TYPE "UDT_UPSMACHSTAT"
TITLE = UDT_MACHSTAT
VERSION : 0.1
//User-defined structure of UPS machine statuses.
   STRUCT
      OpsNormal : Struct   // Ops/Normal
         StopMCP : Bool;   // Byte 1, Bit 0 - Operator Stop MCP Panel
         StopRemoteCon1 : Bool;   // Byte 1, Bit 1 - Operator Stop Remote Console 1
         StopRemoteCon2 : Bool;   // Byte 1, Bit 2 - Operator Stop Remote Console 2
         BuildingStop : Bool;   // Byte 1, Bit 3 - Building Stop via HMI
         BuildingBreak : Bool;   // Byte 1, Bit 4 - Building Break Time via HMI
         PowerSaveShutdown : Bool;   // Byte 1, Bit 5 - Power Save Shutdown
         SorterNotAtSpeed : Bool;   // Byte 1, Bit 6 - Sorter Not at speed
         MaintenanceSysMode : Bool;   // Byte 1, Bit 7 - System in Maintenance Mode
         Spare_8 : Bool;   // Byte 2, Bit 8 - Future / or Machine Specific (To be identyfied)
         Spare_9 : Bool;   // Byte 2, Bit 9 - Future / or Machine Specific (To be identyfied)
         Spare_10 : Bool;   // Byte 2, Bit 10 - Future / or Machine Specific (To be identyfied)
         Spare_11 : Bool;   // Byte 2, Bit 11 - Future / or Machine Specific (To be identyfied)
         Spare_12 : Bool;   // Byte 2, Bit 12 - Future / or Machine Specific (To be identyfied)
         Spare_13 : Bool;   // Byte 2, Bit 13 - Future / or Machine Specific (To be identyfied)
         Spare_14 : Bool;   // Byte 2, Bit 14 - Future / or Machine Specific (To be identyfied)
         Spare_15 : Bool;   // Byte 2, Bit 15 - Future / or Machine Specific (To be identyfied)
         Spare_16 : Bool;   // Byte 3, Bit 16 - Future / or Machine Specific (To be identyfied)
         Spare_17 : Bool;   // Byte 3, Bit 17 - Future / or Machine Specific (To be identyfied)
         Spare_18 : Bool;   // Byte 3, Bit 18 - Future / or Machine Specific (To be identyfied)
         Spare_19 : Bool;   // Byte 3, Bit 19 - Future / or Machine Specific (To be identyfied)
         Spare_20 : Bool;   // Byte 3, Bit 20 - Future / or Machine Specific (To be identyfied)
         Spare_21 : Bool;   // Byte 3, Bit 21 - Future / or Machine Specific (To be identyfied)
         Spare_22 : Bool;   // Byte 3, Bit 22 - Future / or Machine Specific (To be identyfied)
         Spare_23 : Bool;   // Byte 3, Bit 23 - Future / or Machine Specific (To be identyfied)
         Spare_24 : Bool;   // Byte 4, Bit 24 - Future / or Machine Specific (To be identyfied)
         Spare_25 : Bool;   // Byte 4, Bit 25 - Future / or Machine Specific (To be identyfied)
         Spare_26 : Bool;   // Byte 4, Bit 26 - Future / or Machine Specific (To be identyfied)
         Spare_27 : Bool;   // Byte 4, Bit 27 - Future / or Machine Specific (To be identyfied)
         Spare_28 : Bool;   // Byte 4, Bit 28 - Future / or Machine Specific (To be identyfied)
         Spare_29 : Bool;   // Byte 4, Bit 29 - Future / or Machine Specific (To be identyfied)
         Spare_30 : Bool;   // Byte 4, Bit 30 - Future / or Machine Specific (To be identyfied)
         Spare_31 : Bool;   // Byte 4, Bit 31 - Future / or Machine Specific (To be identyfied)
      END_STRUCT;
      SafetyFaults : Struct   // Safety faults
         BuildingEStop : Bool;   // Byte 5, Bit 0 - Building Emergency Stop
         SystemEStop : Bool;   // Byte 5, Bit 1 - System Emergency Stop
         EmerPullCord : Bool;   // Byte 5, Bit 2 - Emergency Pull Cord
         PhotoEyeBlock1 : Bool;   // Byte 5, Bit 3 - Safety Photo Eye Blocked (Long Range Photo Eye) 1
         PlatformLockout1 : Bool;   // Byte 5, Bit 4 - Platform Lockout 1
         PlatformLockout2 : Bool;   // Byte 5, Bit 5 - Platform Lockout 2
         PhotoEyeBlock2 : Bool;   // Byte 5, Bit 6 - Safety Photo Eye Blocked (Long Range Photo Eye) 2
         PhotoEyeBlock3 : Bool;   // Byte 5, Bit 7 - Safety Photo Eye Blocked (Long Range Photo Eye) 3
         Spare_8 : Bool;   // Byte 6, Bit 8 - Future / or Machine Specific (To be identyfied)
         Spare_9 : Bool;   // Byte 6, Bit 9 - Future / or Machine Specific (To be identyfied)
         Spare_10 : Bool;   // Byte 6, Bit 10 - Future / or Machine Specific (To be identyfied)
         Spare_11 : Bool;   // Byte 6, Bit 11 - Future / or Machine Specific (To be identyfied)
         Spare_12 : Bool;   // Byte 6, Bit 12 - Future / or Machine Specific (To be identyfied)
         Spare_13 : Bool;   // Byte 6, Bit 13 - Future / or Machine Specific (To be identyfied)
         Spare_14 : Bool;   // Byte 6, Bit 14 - Future / or Machine Specific (To be identyfied)
         Spare_15 : Bool;   // Byte 6, Bit 15 - Future / or Machine Specific (To be identyfied)
         Spare_16 : Bool;   // Byte 7, Bit 16 - Future / or Machine Specific (To be identyfied)
         Spare_17 : Bool;   // Byte 7, Bit 17 - Future / or Machine Specific (To be identyfied)
         Spare_18 : Bool;   // Byte 7, Bit 18 - Future / or Machine Specific (To be identyfied)
         Spare_19 : Bool;   // Byte 7, Bit 19 - Future / or Machine Specific (To be identyfied)
         Spare_20 : Bool;   // Byte 7, Bit 20 - Future / or Machine Specific (To be identyfied)
         Spare_21 : Bool;   // Byte 7, Bit 21 - Future / or Machine Specific (To be identyfied)
         Spare_22 : Bool;   // Byte 7, Bit 22 - Future / or Machine Specific (To be identyfied)
         Spare_23 : Bool;   // Byte 7, Bit 23 - Future / or Machine Specific (To be identyfied)
         Spare_24 : Bool;   // Byte 8, Bit 24 - Future / or Machine Specific (To be identyfied)
         Spare_25 : Bool;   // Byte 8, Bit 25 - Future / or Machine Specific (To be identyfied)
         Spare_26 : Bool;   // Byte 8, Bit 26 - Future / or Machine Specific (To be identyfied)
         Spare_27 : Bool;   // Byte 8, Bit 27 - Future / or Machine Specific (To be identyfied)
         Spare_28 : Bool;   // Byte 8, Bit 28 - Future / or Machine Specific (To be identyfied)
         Spare_29 : Bool;   // Byte 8, Bit 29 - Future / or Machine Specific (To be identyfied)
         Spare_30 : Bool;   // Byte 8, Bit 30 - Future / or Machine Specific (To be identyfied)
         Spare_31 : Bool;   // Byte 8, Bit 31 - Future / or Machine Specific (To be identyfied)
      END_STRUCT;
      SystemFaults : Struct   // System faults
         PLCRackFault : Bool;   // Byte 9, Bit 0 - PLC Rack Fault
         EncoderFault : Bool;   // Byte 9, Bit 1 - Encoder Fault
         TipperOrDiverterFault : Bool;   // Byte 9, Bit 2 - Tipper / Diverter Fault
         TCPConFail : Bool;   // Byte 9, Bit 3 - TCP Connection Failure
         SensorJam : Bool;   // Byte 9, Bit 4 - Package Detect Sensor Jam
         CamOrScanFail : Bool;   // Byte 9, Bit 5 - Camera / Scanner Failure
         InductPEJam : Bool;   // Byte 9, Bit 6 - Induct Photo Eye Jam
         SortVerificationPEJam : Bool;   // Byte 9, Bit 7 - Sort Verification Photo Eye Jam
         TakeAwayConvPEJam : Bool;   // Byte 10, Bit 8 - Take Away Conveyor Photo Eye Jam
         SorterMechFault : Bool;   // Byte 10, Bit 9 - Sorter Mechanical Fault
         Spare_10 : Bool;   // Byte 10, Bit 10 - Future / or Machine Specific (To be identyfied)
         SorterJam : Bool;   // Byte 10, Bit 11 - Sorter Jam (Logical Failure)
         InductPCAlignmentError : Bool;   // Byte 10, Bit 12 - Induct Photo Cell Alignment Error
         MotorFault : Bool;   // Byte 10, Bit 13 - Motor Fault
         PowerFault : Bool;   // Byte 10, Bit 14 - Power Fault
         Spare_15 : Bool;   // Byte 10, Bit 15 - Future / or Machine Specific (To be identyfied)
         IOComError : Bool;   // Byte 11, Bit 16 - I/O Communications Error
         RemoteIOComError : Bool;   // Byte 11, Bit 17 - Remote I/O Communications Error
         XLeChatComError : Bool;   // Byte 11, Bit 18 - XLe chat Communications Error
         SerialComError : Bool;   // Byte 11, Bit 19 - Serial Communications Error
         SubsystemError : Bool;   // Byte 11, Bit 20 - Subsytem Error (Scale, Camera, etc...)
         VDFFault : Bool;   // Byte 11, Bit 21 - VDF Fault
         SystemResetInitiated : Bool;   // Byte 11, Bit 22 - System Reset Initiated
         PFCStopMode : Bool;   // Byte 11, Bit 23 - PFC not in Run Mode
         NoHitPoints : Bool;   // Byte 12, Bit 24 - No Hit points / Divert Set Ponts found
         MissingTraysDetected : Bool;   // Byte 12, Bit 25 - Missing Trays Detected
         DataFault : Bool;   // Byte 12, Bit 26 - Data Fault, X number of sequential missing valid SORT messages
         Spare_27 : Bool;   // Byte 12, Bit 27 - Future / or Machine Specific (To be identyfied)
         Spare_28 : Bool;   // Byte 12, Bit 28 - Future / or Machine Specific (To be identyfied)
         Spare_29 : Bool;   // Byte 12, Bit 29 - Future / or Machine Specific (To be identyfied)
         Spare_30 : Bool;   // Byte 12, Bit 30 - Future / or Machine Specific (To be identyfied)
         Spare_31 : Bool;   // Byte 12, Bit 31 - Future / or Machine Specific (To be identyfied)
      END_STRUCT;
      OtherFaults : Struct   // Other faults
         ConsoleDisconnect : Bool;   // Byte 13, Bit 0 - Console Disconnect
         PLCChassisPower : Bool;   // Byte 13, Bit 1 - PLC Chassis Power
         SystemInputPower : Bool;   // Byte 13, Bit 2 - System Input Power
         SystemPowerOutput : Bool;   // Byte 13, Bit 3 - System Power Output
         DiverterTipperPower : Bool;   // Byte 13, Bit 4 - Diverter / Tipper Power
         VFDServoFault : Bool;   // Byte 13, Bit 5 - VFD / Servo Fault
         MotorStarterFault : Bool;   // Byte 13, Bit 6 - Motor Starter Fault
         PLCFault : Bool;   // Byte 13, Bit 7 - PLC Fault
         Spare_8 : Bool;   // Byte 14, Bit 8 - Future / or Machine Specific (To be identyfied)
         Spare_9 : Bool;   // Byte 14, Bit 9 - Future / or Machine Specific (To be identyfied)
         Spare_10 : Bool;   // Byte 14, Bit 10 - Future / or Machine Specific (To be identyfied)
         Spare_11 : Bool;   // Byte 14, Bit 11 - Future / or Machine Specific (To be identyfied)
         Spare_12 : Bool;   // Byte 14, Bit 12 - Future / or Machine Specific (To be identyfied)
         Spare_13 : Bool;   // Byte 14, Bit 13 - Future / or Machine Specific (To be identyfied)
         Spare_14 : Bool;   // Byte 14, Bit 14 - Future / or Machine Specific (To be identyfied)
         Spare_15 : Bool;   // Byte 14, Bit 15 - Future / or Machine Specific (To be identyfied)
         Spare_16 : Bool;   // Byte 15, Bit 16 - Future / or Machine Specific (To be identyfied)
         Spare_17 : Bool;   // Byte 15, Bit 17 - Future / or Machine Specific (To be identyfied)
         Spare_18 : Bool;   // Byte 15, Bit 18 - Future / or Machine Specific (To be identyfied)
         Spare_19 : Bool;   // Byte 15, Bit 19 - Future / or Machine Specific (To be identyfied)
         Spare_20 : Bool;   // Byte 15, Bit 20 - Future / or Machine Specific (To be identyfied)
         Spare_21 : Bool;   // Byte 15, Bit 21 - Future / or Machine Specific (To be identyfied)
         Spare_22 : Bool;   // Byte 15, Bit 22 - Future / or Machine Specific (To be identyfied)
         Spare_23 : Bool;   // Byte 15, Bit 23 - Future / or Machine Specific (To be identyfied)
         Spare_24 : Bool;   // Byte 16, Bit 24 - Future / or Machine Specific (To be identyfied)
         Spare_25 : Bool;   // Byte 16, Bit 25 - Future / or Machine Specific (To be identyfied)
         Spare_26 : Bool;   // Byte 16, Bit 26 - Future / or Machine Specific (To be identyfied)
         Spare_27 : Bool;   // Byte 16, Bit 27 - Future / or Machine Specific (To be identyfied)
         Spare_28 : Bool;   // Byte 16, Bit 28 - Future / or Machine Specific (To be identyfied)
         Spare_29 : Bool;   // Byte 16, Bit 29 - Future / or Machine Specific (To be identyfied)
         Spare_30 : Bool;   // Byte 16, Bit 30 - Future / or Machine Specific (To be identyfied)
         Spare_31 : Bool;   // Byte 16, Bit 31 - Future / or Machine Specific (To be identyfied)
      END_STRUCT;
   END_STRUCT;

END_TYPE

TYPE "UDT_UPS1stStageFlowControlConfiguration"
VERSION : 0.1
   STRUCT
      NumberOfInfeedsInUse : Int;   // Number of infeeds used
      ThresholdConsecutivesAboveSP : Int;   // Number of consecutive intervals above set point to trigger flow control
      ThresholdConsecutivesBelowSP : Int;   // Number of consecutive intervals below set point to reset flow control
      IntervalsNumberOfEvaluationPeriod : Int;   // Number of intervals for evaluation of flow control
      LegthBasedFlowControl : Bool;   // TRUE = The input of the counts is length FALSE = The input is counts of parcel
      IsLengthImperial : Bool;   // TRUE =  Length is given in inches. FALSE = Lentgh is given in mm
      IncrementingCounts : Bool;   // TRUE = Input data are incremented. FALSE =  Input data are updated every 15 sec
      Infeed : Array[1..10] of Struct
         RegisterOffset : Int;   // Number of register offset for evalueated flow calculation
         MinimumTimeToStop : UInt;   // Minimum stop time of divert
         IsHighPriority : Bool;   // TRUE= The divert is high priority
         IsNotAllowedToStop : Bool;   // TRUE= The divert is not allowed to stop (e.g. Recirculation)
      END_STRUCT;
   END_STRUCT;

END_TYPE

TYPE "UDT_UPSLostCounters"
VERSION : 0.1
   STRUCT
      LostInTracking : DInt;   // Parcel lost in tracking
      NoUPSID : DInt;   // No UPS ID created (missing SCAN_DATA_2)
      NoSortRcv : DInt;   // No sort instruction
   END_STRUCT;

END_TYPE

FUNCTION "FC_CharToInt" : Void
TITLE = FC_TimeToString
{ S7_Optimized_Access := 'TRUE' }
AUTHOR : MHSE
FAMILY : GeneralSystemFunctions
VERSION : 3.0
// ATTRIBUTES
// AUTO_NUMBER = True
// BLOCK_NUMBER = 32
// END_ATTRIBUTES
//Function to convert date in DTL to the string format.
   VAR_INPUT
      Offset : Int;   // Offset in Char Data
      Data : "UDT_Message";
   END_VAR

   VAR_OUTPUT
      qi_data : Int;   // Int format data
   END_VAR


BEGIN


	(*
	----------------------------------------------------------------------------------------
	|                                                                                      |
	|  Copyright  2019             MHS                                                     |
	|  All Rights Reserved         Larenweg 90                                             |
	|                              5234 KC 's-Hertogenbosch,                               |
	|                              Netherlands                                             |
	|                                                                                      |
	----------------------------------------------------------------------------------------

	Version history:
	Date        | Version   | Author       | Remark
	----------------------------------------------------------------------------------------
	28/05/2021  | 0.1       | M. Jager      | first release MHS TIA 16.0

	*)

	#qi_data :=
	(STRING_TO_INT(IN := (CHAR_TO_STRING(IN := #Data.Character[#Offset]))) * 1000) +
	(STRING_TO_INT(IN := (CHAR_TO_STRING(IN := #Data.Character[#Offset + 1]))) * 100) +
	(STRING_TO_INT(IN := (CHAR_TO_STRING(IN := #Data.Character[#Offset + 2]))) * 10) +
	(STRING_TO_INT(IN := (CHAR_TO_STRING(IN := #Data.Character[#Offset + 3]))));
END_FUNCTION

TYPE "UDT_ConveyorHandshake"
TITLE = UDT_ConveyorHandshake
VERSION : 0.1
//User-defined structure of conveyor handshake variables.
   STRUCT
      GIN : Int;   // General identification number
      NrOfPosToShift : Int;   // Number of positions to shift
      DownstreamDisplacement : Int;   // Displacement from downstream [cm]
      RTS { ExternalAccessible := 'False'; ExternalVisible := 'False'; ExternalWritable := 'False'} : Bool;   // Conveyor ready to send
      RTR { ExternalAccessible := 'False'; ExternalVisible := 'False'; ExternalWritable := 'False'} : Bool;   // Conveyor ready to receive
      TIP { ExternalAccessible := 'False'; ExternalVisible := 'False'; ExternalWritable := 'False'} : Bool;   // Transfer in progress
      ResetEnergySave { ExternalAccessible := 'False'; ExternalVisible := 'False'; ExternalWritable := 'False'} : Bool;   // Reset energy save mode
      CascadeStartUp { ExternalAccessible := 'False'; ExternalVisible := 'False'; ExternalWritable := 'False'} : Bool;   // Cascade startup
      ReqStop { ExternalAccessible := 'False'; ExternalVisible := 'False'; ExternalWritable := 'False'} : Bool;   // Request stop
   END_STRUCT;

END_TYPE

FUNCTION "FC_UPSMsgId" : Void
TITLE = FC_MSGID
{ S7_Optimized_Access := 'TRUE' }
AUTHOR : MHSE
FAMILY : UPS_SpecificCommunication
VERSION : 3.0
// ATTRIBUTES
// AUTO_NUMBER = True
// BLOCK_NUMBER = 34
// END_ATTRIBUTES
//Function to create the UPS message ID.
   VAR_INPUT
      is_ActualDateTime : String;   // Actual date and time
      is_ModuleName : String;   // Module type
      is_DeviceNumber : String;   // Device number
   END_VAR

   VAR_IN_OUT
      iqs_MSGID : String;   // MSGID character string
      iqdi_UniqueMsgID : DInt;   // Unique message ID integer value
   END_VAR

   VAR_TEMP
      ts_Timestamp : String;   // Timestamp
      ts_UniqueMsgID : String[11];   // Unique message ID character sting
      ti_UniqueMsgIDLen : Int;   // Unique message ID length
      ti_i : Int;   // Loop counter
   END_VAR

   VAR CONSTANT
      cc_Dash : Char := '-';   // Dash sign
   END_VAR


BEGIN
	(*
	----------------------------------------------------------------------------------------

	Version history:
	Date        | Version   | Author        | Remark
	----------------------------------------------------------------------------------------
	24/05/2019  | 0.1       | L.Klar        | first release MHS TIA 15.1
	24/07/2019  | 2.0       | L.Klar        | 2.0 MHS library release TIA 15.1
	23/08/2019  | 2.1       | K.Pokorski    | Comments simplified
	12/11/2019  | 3.0       | P.Majka       | 3.0 MHS library release TIA 15.1
	21/02/2023  | 4.0       | F.Baten       | 4.0 Release TIA 17.5
	*)

	REGION 1 – Initialization

	    #ts_Timestamp := '';
	    #ti_UniqueMsgIDLen := 0;
	    #ti_i := 0;

	END_REGION

	REGION 2 – Timestamp preparation

	    #ts_Timestamp := RIGHT(IN := #is_ActualDateTime, L := 12);

	END_REGION

	REGION 3 – Unique message ID preparation

	    // Unique message ID incrementation
	    IF (#iqdi_UniqueMsgID < 2147483647)     // Unique message ID is lower than 2147483647
	    THEN

	        #iqdi_UniqueMsgID += 1;

	    ELSE

	        #iqdi_UniqueMsgID := 0;

	    END_IF;

	    // Unique message ID character string clearing
	    #ts_UniqueMsgID := '';

	    // Unique message ID integer conversion to a character string
	    VAL_STRG(IN := #iqdi_UniqueMsgID,
	             SIZE := 0,
	             PREC := 0,
	             FORMAT := 0,
	             P := 1,
	             OUT => #ts_UniqueMsgID);

	    // Length of the unique message ID character string
	    #ti_UniqueMsgIDLen := LEN(#ts_UniqueMsgID);

	    // Unique message ID character string leading zeros addition
	    IF (#ti_UniqueMsgIDLen < 11)        // Unique message ID length lower than 11
	    THEN

	        FOR #ti_i := 1 TO 11 - #ti_UniqueMsgIDLen DO

	            #ts_UniqueMsgID := CONCAT(IN1 := '0',
	                                      IN2 := #ts_UniqueMsgID);

	        END_FOR;

	    END_IF;

	END_REGION

	REGION 4 – MSGID preparation

	    #iqs_MSGID := CONCAT(IN1 := #is_ModuleName,      // Module name
	                         IN2 := #cc_Dash,            // Dash sign - "-"
	                         IN3 := #is_DeviceNumber,    // Device number
	                         IN4 := #cc_Dash,            // Dash sign - "-"
	                         IN5 := #ts_Timestamp,       // Timestamp
	                         IN6 := #cc_Dash,            // Dash sign - "-"
	                         IN7 := #ts_UniqueMsgID);    // Unique message ID

	END_REGION
END_FUNCTION

FUNCTION_BLOCK "FB_SickVmsTcpipReceive"
TITLE = FB_TCPIPReceive
{ S7_Optimized_Access := 'TRUE' }
AUTHOR : MHSE
FAMILY : Communication
VERSION : 3.0
// ATTRIBUTES
// AUTO_NUMBER = True
// BLOCK_NUMBER = 45
// END_ATTRIBUTES
//Function block to receive data from TCPIP.
   VAR_INPUT
      i_UDT_Connection { ExternalAccessible := 'False'; ExternalVisible := 'False'; ExternalWritable := 'False'} : "UDT_Connection";   // Connection parameters
      ix_EnableReceive { ExternalAccessible := 'False'; ExternalVisible := 'False'; ExternalWritable := 'False'} : Bool;   // Enable receive
   END_VAR

   VAR_OUTPUT
      qx_Error { ExternalAccessible := 'False'; ExternalVisible := 'False'; ExternalWritable := 'False'} : Bool;   // Collective error output
      qx_Warning { ExternalAccessible := 'False'; ExternalVisible := 'False'; ExternalWritable := 'False'} : Bool;   // Collective warning output
   END_VAR

   VAR_IN_OUT
      iq_UDT_FifoHeader : "UDT_FifoHeader";   // Fifo header
      iqs_FifoData : Array[*] of "UDT_Message";   // Fifo data
      iq_UDT_Statistics : "UDT_TCPIPReceiveStatistics";   // Statistic structure
   END_VAR

   VAR
      s_FB_TRCV {InstructionName := 'TRCV'; LibVersion := '4.0'; ExternalAccessible := 'False'; ExternalVisible := 'False'; ExternalWritable := 'False'; S7_SetPoint := 'False'} : TRCV;   // Siemens "TRCV" block - to receive the data from TCPIP socket
      ss_TRCV { ExternalAccessible := 'False'; ExternalVisible := 'False'; ExternalWritable := 'False'} : Struct   // TRCV block interface structure
         Enable { ExternalAccessible := 'False'; ExternalVisible := 'False'; ExternalWritable := 'False'} : Bool;   //    TRCV - Enable
         NDR { ExternalAccessible := 'False'; ExternalVisible := 'False'; ExternalWritable := 'False'} : Bool;   //    TRCV - New data available
         Busy { ExternalAccessible := 'False'; ExternalVisible := 'False'; ExternalWritable := 'False'} : Bool;   //    TRCV - Busy
         Error { ExternalAccessible := 'False'; ExternalVisible := 'False'; ExternalWritable := 'False'} : Bool;   //    TRCV - Error
         Status { ExternalAccessible := 'False'; ExternalVisible := 'False'; ExternalWritable := 'False'} : Word;   //    TRCV - Status
         RcvLen { ExternalAccessible := 'False'; ExternalVisible := 'False'; ExternalWritable := 'False'} : UDInt;   //    TRCV - Received length
         Data { ExternalAccessible := 'False'; ExternalVisible := 'False'; ExternalWritable := 'False'} : Array[0..999] of Char;   //    TRCV - Data
      END_STRUCT;
      s_UDT_MsgArray { ExternalAccessible := 'False'; ExternalVisible := 'False'; ExternalWritable := 'False'; S7_SetPoint := 'False'} : "UDT_Message";   // Message character array
      s_UDT_MsgPartArray { ExternalAccessible := 'False'; ExternalVisible := 'False'; ExternalWritable := 'False'; S7_SetPoint := 'False'} : "UDT_Message";   // Part of the message character array
      ss_Status { ExternalAccessible := 'False'; ExternalVisible := 'False'; ExternalWritable := 'False'} : Struct   // Status structure
         ErrorCode { ExternalAccessible := 'False'; ExternalVisible := 'False'; ExternalWritable := 'False'} : Struct   // Error code structure
            TRCV { ExternalAccessible := 'False'; ExternalVisible := 'False'; ExternalWritable := 'False'} : Word;   // Siemens TRCV error code - Check documentation
         END_STRUCT;
         FIFORcvStatus { ExternalAccessible := 'False'; ExternalVisible := 'False'; ExternalWritable := 'False'} : "UDT_FifoStatus";   // Receive FIFO status structure
         FIFORcvError { ExternalAccessible := 'False'; ExternalVisible := 'False'; ExternalWritable := 'False'; S7_SetPoint := 'True'} : Bool;   // Receive FIFO error
         FIFORcvWarning { ExternalAccessible := 'False'; ExternalVisible := 'False'; ExternalWritable := 'False'; S7_SetPoint := 'True'} : Bool;   // Receive  FIFO warning
         ReceiveError { ExternalAccessible := 'False'; ExternalVisible := 'False'; ExternalWritable := 'False'} : Bool;   // TRCV block operation error - Check TRCVStatus
      END_STRUCT;
      sdi_RcvMsgCounter { ExternalAccessible := 'False'; ExternalVisible := 'False'; ExternalWritable := 'False'} : DInt;   // Total received messages counter
      si_RcvMsgOffset { ExternalAccessible := 'False'; ExternalVisible := 'False'; ExternalWritable := 'False'} : Int;   // Received message offset
      si_RcvMsgLen { ExternalAccessible := 'False'; ExternalVisible := 'False'; ExternalWritable := 'False'} : Int;   // Received message length
      si_NrOfRcvMsg { ExternalAccessible := 'False'; ExternalVisible := 'False'; ExternalWritable := 'False'} : Int;   // Number of received messages in one frame
      si_RcvMsgPartLen { ExternalAccessible := 'False'; ExternalVisible := 'False'; ExternalWritable := 'False'} : Int;   // Length of the part of received message
      si_i { ExternalAccessible := 'False'; ExternalVisible := 'False'; ExternalWritable := 'False'} : Int;   // Loop counter
      si_MaxMsgLen { ExternalAccessible := 'False'; ExternalVisible := 'False'; ExternalWritable := 'False'} : Int;   // Maximum message length
      sx_RcvMsgPart { ExternalAccessible := 'False'; ExternalVisible := 'False'; ExternalWritable := 'False'} : Bool;   // Received part of the message
      sx_InvalidTermination { ExternalAccessible := 'False'; ExternalVisible := 'False'; ExternalWritable := 'False'} : Bool;   // Termination sign missing
   END_VAR

   VAR CONSTANT
      cc_CRLF_R : Char := '$03';
      cc_CRLF_L : Char := '$03';   // Last termination sign
      cc_NULL : Char := '$00';   // NULL sign
   END_VAR


BEGIN
	(*
	----------------------------------------------------------------------------------------
	|                                                                                      |
	|  Copyright  2019             MHS                                                     |
	|  All Rights Reserved         Larenweg 90                                             |
	|                              5234 KC 's-Hertogenbosch,                               |
	|                              Netherlands                                             |
	|                                                                                      |
	----------------------------------------------------------------------------------------

	Version history:
	Date        | Version   | Author       | Remark
	----------------------------------------------------------------------------------------
	24/05/2019  | 0.1       | L.Klar       | first release MHS TIA 15.1
	17/06/2019  | 0.3       | A.Nowak      | Replace 2nd level subregions with comments (5.3)
	24/07/2019  | 2.0       | L.Klar       | 2.0 MHS library release TIA 15.1
	22/08/2019  | 2.1       | K.Pokorski   | Comments adjusted
	12/09/2019  | 2.2       | A.Nowak      | Delete buffer size variable
	20/09/2019  | 2.3       | J.Krawczuk   | Replacing UDT_HeartbeatStatus structure to internal structure
	01/10/2019  | 2.4       | A.Nowak      | Implementation of the new FIFO block
	12/11/2019  | 3.0       | P.Majka      | 3.0 MHS library release TIA 15.1
	23/03/2021  | 3.1       | L.Klar       | Static variables data types changed form uint to int
	14/08/2021  | 3.2       | S. Deulkar   | In region 5.3, conveted variable to ULINT because it was giving warning
	14/03/2024  | 4.1       | S. Nieswiec  | Added from Hannover project and changed name according to standard
	02/05/2024  | 4.2       | J.Majer      | Datatype conversions changed from automatic to explicit, to accomodate IEC 61131-3 standard
	*)

	REGION 1 – Update FIFO header status bits

	    // Mode 'S' - FIFO register status update
	    "FC_Fifo"(ic_Mode := 'S',
	              qUDT_Status => #ss_Status.FIFORcvStatus,
	              qx_Error => #ss_Status.FIFORcvError,
	              qx_Warning => #ss_Status.FIFORcvWarning,
	              iqv_Data := #s_UDT_MsgArray,
	              iqUDT_FifoHeader := #iq_UDT_FifoHeader,
	              iqv_DataBuffer := #iqs_FifoData);


	END_REGION

	REGION 2 – Maximum number of message arrays elements

	    #si_MaxMsgLen := "FC_GetNrOfArrayEl"(iv_Array := #s_UDT_MsgArray.Character);

	END_REGION

	REGION 3 – Receive enable

	    // Allow receiving if the connection is established and there are no fifo errors
	    #ss_TRCV.Enable :=
	    #ix_EnableReceive
	    AND NOT #ss_Status.FIFORcvError;

	END_REGION

	REGION 4 – Receive data

	    // Data received in an ADHOC mode - data available immediately
	    #s_FB_TRCV(EN_R := #ss_TRCV.Enable,
	               ID := #i_UDT_Connection.ID,
	               LEN := 0,
	               ADHOC := TRUE,
	               NDR => #ss_TRCV.NDR,
	               BUSY => #ss_TRCV.Busy,
	               ERROR => #ss_TRCV.Error,
	               STATUS => #ss_TRCV.Status,
	               RCVD_LEN => #ss_TRCV.RcvLen,
	               DATA := #ss_TRCV.Data);

	END_REGION

	IF #ss_TRCV.RcvLen > 1000 THEN
	    #ss_TRCV.RcvLen := 1000;
	END_IF;

	REGION 5 – Received data handling

	    // Receiving data was successful
	    IF (#ss_TRCV.NDR                    // New data received without error
	        AND NOT #ss_TRCV.Busy           // Job not yet started or already completed
	        AND NOT #ss_TRCV.Error          // No errors during receiving messages
	        AND #ss_TRCV.RcvLen > 0)        // Length greater than zero
	    THEN

	        REGION 5.1 – Initialization

	            #si_RcvMsgLen := 0;
	            #si_RcvMsgOffset := 0;
	            #si_NrOfRcvMsg := 0;

	        END_REGION

	        REGION 5.2 – Received part of the message

	            // Move part of the messages to a buffer if available
	            IF (#sx_RcvMsgPart)                             // Message part available
	            THEN

	                #s_UDT_MsgArray := #s_UDT_MsgPartArray;
	                #sx_RcvMsgPart := FALSE;

	            END_IF;

	        END_REGION

	        REGION 5.3 – Message handling

	            FOR #si_i := 0 TO UDINT_TO_INT(#ss_TRCV.RcvLen) - 1 DO

	                // Message length validation
	                IF (#si_RcvMsgLen + #si_RcvMsgPartLen < #si_MaxMsgLen)
	                THEN

	                    // Termination sign found
	                    IF (#ss_TRCV.Data[#si_i] = #cc_CRLF_R)
	                    THEN

	                        // Move received message to the message array
	                        MOVE_BLK(IN := #ss_TRCV.Data[#si_RcvMsgOffset],
	                                 COUNT := INT_TO_ULINT(#si_RcvMsgLen + 1),
	                                 OUT => #s_UDT_MsgArray.Character[#si_RcvMsgPartLen]);

	                        // Clear NOT used message array characters
	                        FILL_BLK(IN := #cc_NULL,
	                                 COUNT := INT_TO_ULINT(#si_MaxMsgLen - #si_RcvMsgLen + #si_RcvMsgPartLen - 1),
	                                 OUT => #s_UDT_MsgArray.Character[#si_RcvMsgLen + #si_RcvMsgPartLen + 1]);

	                        // Check and clear termination sign
	                        IF (#si_RcvMsgLen + #si_RcvMsgPartLen - 1) >= 0 AND (#si_RcvMsgLen + #si_RcvMsgPartLen - 1) < #si_MaxMsgLen THEN
	                            IF (#s_UDT_MsgArray.Character[#si_RcvMsgLen + #si_RcvMsgPartLen] = #cc_CRLF_R)        // Character is a termination sign
	                            THEN
	                                #sx_InvalidTermination := FALSE;                                    // Reset the invalid termination bit

	                                // Termination sign invalid - error generated, statistics increased
	                            ELSE

	                                #sx_InvalidTermination := TRUE;
	                                #iq_UDT_Statistics.InvalidMsg += 1;

	                            END_IF;
	                        ELSE
	                            #iq_UDT_Statistics.InvalidMsg += 1;
	                        END_IF;


	                        // Move message into the FIFO data block
	                        IF (NOT #sx_InvalidTermination)                                         // No termination sign error
	                        THEN

	                            // Mode 'W' - Write FIFO record
	                            "FC_Fifo"(ic_Mode := 'W',
	                                      qUDT_Status => #ss_Status.FIFORcvStatus,
	                                      qx_Error => #ss_Status.FIFORcvError,
	                                      qx_Warning => #ss_Status.FIFORcvWarning,
	                                      iqv_Data := #s_UDT_MsgArray,
	                                      iqUDT_FifoHeader := #iq_UDT_FifoHeader,
	                                      iqv_DataBuffer := #iqs_FifoData);


	                        END_IF;


	                        // Update lengths and counters
	                        #si_RcvMsgPartLen := 0;
	                        #si_RcvMsgOffset += #si_RcvMsgLen + 1;
	                        #si_RcvMsgLen := 0;
	                        #si_NrOfRcvMsg += 1;
	                        #sdi_RcvMsgCounter += 1;

	                        // Termination sign not found
	                    ELSE

	                        #si_RcvMsgLen := #si_RcvMsgLen + 1;                               // Increment received message length

	                    END_IF;

	                    // Message length invalid - reset message length and increase statistics
	                ELSE

	                    #si_RcvMsgLen := 0;
	                    #iq_UDT_Statistics.InvalidMsg += 1;

	                END_IF;

	            END_FOR;

	        END_REGION

	        REGION 5.4 – Part of the message preparation

	            // Move part of the message to buffer when last received sign is not a termination signs
	            IF (#ss_TRCV.Data[UDINT_TO_INT(#ss_TRCV.RcvLen) - 1] <> #cc_CRLF_R            // Last received sign is not a termination sing
	                AND #si_RcvMsgLen < #si_MaxMsgLen)                         // Message length valid
	            THEN

	                // Fill not used message char array elements with '$00'
	                FILL_BLK(IN := '$00',
	                         COUNT := INT_TO_ULINT(#si_MaxMsgLen) -
	                         INT_TO_ULINT(#si_RcvMsgLen),
	                         OUT => #s_UDT_MsgPartArray.Character[#si_RcvMsgLen]);

	                // Move part of the message to a buffer
	                MOVE_BLK(IN := #ss_TRCV.Data[#si_RcvMsgOffset],
	                         COUNT := INT_TO_ULINT(#si_RcvMsgLen),
	                         OUT => #s_UDT_MsgPartArray.Character[0]);

	                // Set the part of the message received bit and move length of the received message into the length of the part of the message variable
	                #sx_RcvMsgPart := TRUE;
	                #si_RcvMsgPartLen := #si_RcvMsgLen;

	            END_IF;

	        END_REGION

	    END_IF;

	END_REGION

	REGION 6 – Status

	    REGION 6.1 - Block status

	        // Receive error
	        #ss_Status.ReceiveError := #ss_TRCV.Error;

	        // Parametrization collective error output
	        #qx_Error :=
	        #ss_Status.FIFORcvError                          // FIFO error
	        OR #ss_Status.ReceiveError;                      // Receive error

	        // Parametrization collective warning output
	        #qx_Warning := #ss_Status.FIFORcvWarning;        // FIFO warning

	    END_REGION

	    REGION 6.2 - Error code preparation

	        IF (#ss_TRCV.#Status > 16#8000
	            OR #ss_TRCV.#Status = 16#0)
	        THEN

	            #ss_Status.ErrorCode.TRCV := #ss_TRCV.#Status;

	        END_IF;

	    END_REGION

	END_REGION
END_FUNCTION_BLOCK

FUNCTION_BLOCK "FB_TCPIPConnect"
TITLE = FB_TCPIPConnect
{ S7_Optimized_Access := 'TRUE' }
AUTHOR : MHSE
FAMILY : Communication
VERSION : 3.0
// ATTRIBUTES
// AUTO_NUMBER = True
// BLOCK_NUMBER = 231
// END_ATTRIBUTES
//Function block to establish and terminateTCPIP connection.
   VAR_INPUT
      iUDT_Connection { ExternalAccessible := 'False'; ExternalVisible := 'False'; ExternalWritable := 'False'} : "UDT_Connection";   // Connection parameters
   END_VAR

   VAR_OUTPUT
      qUDT_HMIStatus { ExternalAccessible := 'False'; ExternalVisible := 'False'; ExternalWritable := 'False'} : "UDT_TCPIPConnectStatus";   // HMI status structure
      qUDT_Status { ExternalAccessible := 'False'; ExternalVisible := 'False'; ExternalWritable := 'False'} : "UDT_CommonStatus";   // Common status structure
      qx_Connected { ExternalAccessible := 'False'; ExternalVisible := 'False'; ExternalWritable := 'False'} : Bool;   // Connected status
   END_VAR

   VAR_IN_OUT
      iqUDT_EquipmentControl : "UDT_EquipmentControl";   // Equipment control structure
      iqUDT_Statistics : "UDT_TCPIPConnectStatistics";   // Statistic structure
      iqx_Reconnect { ExternalAccessible := 'False'; ExternalVisible := 'False'; ExternalWritable := 'False'} : Bool;   // Reconnect command
   END_VAR

   VAR
      sUDT_CommonStatus { ExternalAccessible := 'False'; ExternalVisible := 'False'; ExternalWritable := 'False'; S7_SetPoint := 'False'} : "UDT_CommonStatus";   // Common status structure
      sFB_TCON {InstructionName := 'TCON'; LibVersion := '4.0'; ExternalAccessible := 'False'; ExternalVisible := 'False'; ExternalWritable := 'False'; S7_SetPoint := 'False'} : TCON;   // Siemens "TCON" block - to establish the connection
      sFB_TDISCON {InstructionName := 'TDISCON'; LibVersion := '2.1'; ExternalAccessible := 'False'; ExternalVisible := 'False'; ExternalWritable := 'False'; S7_SetPoint := 'False'} : TDISCON;   // Siemens "TDISCON" block - to terminate the connection
      sFB_DIAG {InstructionName := 'T_DIAG'; LibVersion := '1.2'; ExternalAccessible := 'False'; ExternalVisible := 'False'; ExternalWritable := 'False'; S7_SetPoint := 'False'} : T_DIAG;   // Siemens "T_DIAG" block - to diagnose the connection
      sFB_TimerConTimeout { ExternalAccessible := 'False'; ExternalVisible := 'False'; ExternalWritable := 'False'; S7_SetPoint := 'False'} : "FB_TimerOnOffDelay";   // MHS "FB_TimerOnOffDelay" block - to measure the connection timeout
      sFB_TimerFilter { ExternalAccessible := 'False'; ExternalVisible := 'False'; ExternalWritable := 'False'; S7_SetPoint := 'False'} : "FB_TimerOnOffDelay";   // MHS "FB_TimerOnOffDelay" block - to filter the connection established signal
      sv_InterfaceData {InstructionName := 'TCON_IP_v4'; LibVersion := '1.0'; ExternalAccessible := 'False'; ExternalVisible := 'False'; ExternalWritable := 'False'; S7_SetPoint := 'False'} : TCON_IP_v4;   // TCON Interface configuration data
      sR_TRIG_ConnectionLost {InstructionName := 'R_TRIG'; LibVersion := '1.0'; ExternalAccessible := 'False'; ExternalVisible := 'False'; ExternalWritable := 'False'; S7_SetPoint := 'False'} : R_TRIG;   // Siemens "R_TRIG" - to prepare rising edge signal on Connection lost signal
      sR_TRIG_Reset {InstructionName := 'R_TRIG'; LibVersion := '1.0'; ExternalAccessible := 'False'; ExternalVisible := 'False'; ExternalWritable := 'False'; S7_SetPoint := 'False'} : R_TRIG;   // Siemens "R_TRIG" - to prepare rising edge signal on reset data signal
      sa_Connect { ExternalAccessible := 'False'; ExternalVisible := 'False'; ExternalWritable := 'False'} : Struct   // TCON interface structure
         Request { ExternalAccessible := 'False'; ExternalVisible := 'False'; ExternalWritable := 'False'} : Bool;   //  TCON - Request
         Done { ExternalAccessible := 'False'; ExternalVisible := 'False'; ExternalWritable := 'False'} : Bool;   //  TCON - Done
         Busy { ExternalAccessible := 'False'; ExternalVisible := 'False'; ExternalWritable := 'False'} : Bool;   //  TCON - Busy
         Error { ExternalAccessible := 'False'; ExternalVisible := 'False'; ExternalWritable := 'False'} : Bool;   //  TCON - Error
         Active { ExternalAccessible := 'False'; ExternalVisible := 'False'; ExternalWritable := 'False'} : Bool;   //  TCON - Active
         Status { ExternalAccessible := 'False'; ExternalVisible := 'False'; ExternalWritable := 'False'} : Word;   //  TCON - Status
      END_STRUCT;
      sa_Disconnect { ExternalAccessible := 'False'; ExternalVisible := 'False'; ExternalWritable := 'False'} : Struct   // TDISCON interface structure
         Request { ExternalAccessible := 'False'; ExternalVisible := 'False'; ExternalWritable := 'False'} : Bool;   //  TDISCON - Request
         Done { ExternalAccessible := 'False'; ExternalVisible := 'False'; ExternalWritable := 'False'} : Bool;   //  TDISCON - Done
         Busy { ExternalAccessible := 'False'; ExternalVisible := 'False'; ExternalWritable := 'False'} : Bool;   //  TDISCON - Busy
         Error { ExternalAccessible := 'False'; ExternalVisible := 'False'; ExternalWritable := 'False'} : Bool;   //  TDISCON - Error
         Active { ExternalAccessible := 'False'; ExternalVisible := 'False'; ExternalWritable := 'False'} : Bool;   //  TDISCON - Active
         Status { ExternalAccessible := 'False'; ExternalVisible := 'False'; ExternalWritable := 'False'} : Word;   //  TDISCON - Status
      END_STRUCT;
      sa_Diag { ExternalAccessible := 'False'; ExternalVisible := 'False'; ExternalWritable := 'False'} : Struct   // T_DIAG block diagnostic variables
         Request { ExternalAccessible := 'False'; ExternalVisible := 'False'; ExternalWritable := 'False'} : Bool;   //  TDIAG - Request
         Done { ExternalAccessible := 'False'; ExternalVisible := 'False'; ExternalWritable := 'False'} : Bool;   //  TDIAG - Done
         Busy { ExternalAccessible := 'False'; ExternalVisible := 'False'; ExternalWritable := 'False'} : Bool;   //  TDIAG - Busy
         Error { ExternalAccessible := 'False'; ExternalVisible := 'False'; ExternalWritable := 'False'} : Bool;   //  TDIAG - Error
         Active { ExternalAccessible := 'False'; ExternalVisible := 'False'; ExternalWritable := 'False'} : Bool;   //  TDIAG - Active
         Status { ExternalAccessible := 'False'; ExternalVisible := 'False'; ExternalWritable := 'False'} : Word;   //  TDIAG - Status
         Result {InstructionName := 'TDiag_Status'; LibVersion := '1.0'; ExternalAccessible := 'False'; ExternalVisible := 'False'; ExternalWritable := 'False'} : TDiag_Status;   //  TDIAG - Result
      END_STRUCT;
      sx_Connected { ExternalAccessible := 'False'; ExternalVisible := 'False'; ExternalWritable := 'False'} : Bool;   // Connection established memory
      sx_ConnectedFiltred { ExternalAccessible := 'False'; ExternalVisible := 'False'; ExternalWritable := 'False'} : Bool;   // Connection established memory (filtred)
      sx_CommunicationFault { ExternalAccessible := 'False'; ExternalVisible := 'False'; ExternalWritable := 'False'} : Bool;   // Communication fault
   END_VAR


BEGIN
	(*
	----------------------------------------------------------------------------------------

	Version history:
	Date        | Version   | Author        | Remark
	----------------------------------------------------------------------------------------
	24/05/2019  | 0.1       | L.Klar        | first release MHS TIA 15.1
	13/06/2019  | 0.2       | A.Nowak       | Delete writing to variable - S_FB_Timer_ConTimeout
	24/06/2019  | 0.3       | L.Klar        | Status running added
	25/06/2019  | 0.5       | L.Klar        | Statistics changed to InOut
	24/07/2019  | 2.0       | L.Klar        | 2.0 MHS library release TIA 15.1
	21/08/2019  | 2.1       | K.Pokorski    | Comments adjusted
	26/09/2019  | 2.2       | A.Nowak       | Delete static status structure and change region 9. Create new static sx_CommunicationFault.
	09/10/2019  | 2.3       | M.Kurc        | System equipment control added
	04/11/2019  | 2.4       | L.Klar        | 10 Hz clock and first scan changed from memory bit to DB variable
	19/11/2019  | 2.5       | L.Klar        | Status outputs corrected
	20/11/2019  | 3.0       | P.Majka       | 3.0 MHS library release TIA 15.1
	21/02/2023  | 4.0       | F.Baten       | 4.0 Release TIA 17.5
	*)

	REGION 1 – Initialization

	    // Reset connected status bit and reconnect command bit during first PLC scan
	    IF ("DB_Memory".FirstScan)             // First PLC scan occured
	    THEN

	        #sx_Connected := FALSE;
	        #iqx_Reconnect := TRUE;

	    END_IF;

	END_REGION

	REGION 2 – Connection error reset

	    // Reset errors and blocks statuses when no connection state available and communication fault reset received
	    #sR_TRIG_Reset(CLK := #iqUDT_EquipmentControl.Command.Reset);

	    IF (#sx_CommunicationFault                                      // Communication fault
	        AND #sR_TRIG_Reset.Q)                                      // Reset signal trigger
	    THEN

	        #sa_Connect.Status := 16#0;
	        #sa_Disconnect.Status := 16#0;
	        #sa_Diag.Status := 16#0;
	        #sx_CommunicationFault := FALSE;

	    END_IF;

	END_REGION

	REGION 3 – Communication Interface preparation

	    #sv_InterfaceData.InterfaceId := #iUDT_Connection.Interface_ID;                       // HW-identifier of IE-interface submodule
	    #sv_InterfaceData.ID := #iUDT_Connection.ID;                                          // Connection reference / identifier
	    #sv_InterfaceData.ConnectionType := 16#0B;                                             // Type OF connection: 11=TCP/IP, 19=UDP 17=TCP/IP
	    #sv_InterfaceData.ActiveEstablished := #iUDT_Connection.ActiveEstablished;            // Active/passive connection establishment
	    #sv_InterfaceData.RemoteAddress.ADDR[1] := INT_TO_BYTE(#iUDT_Connection.IP[1]);       // Remote IP address (IPv4) - x.0.0.0
	    #sv_InterfaceData.RemoteAddress.ADDR[2] := INT_TO_BYTE(#iUDT_Connection.IP[2]);       // Remote IP address (IPv4) - 0.x.0.0
	    #sv_InterfaceData.RemoteAddress.ADDR[3] := INT_TO_BYTE(#iUDT_Connection.IP[3]);       // Remote IP address (IPv4) - 0.0.x.0
	    #sv_InterfaceData.RemoteAddress.ADDR[4] := INT_TO_BYTE(#iUDT_Connection.IP[4]);       // Remote IP address (IPv4) - 0.0.0.x

	    // Set local or remote port depending on whether the PLC is active or passive device in connection
	    IF (#sv_InterfaceData.ActiveEstablished)                                               // Active connection
	    THEN

	        #sv_InterfaceData.LocalPort := 0;
	        #sv_InterfaceData.RemotePort := #iUDT_Connection."Port";

	        // Passive connection
	    ELSE

	        #sv_InterfaceData.LocalPort := #iUDT_Connection."Port";
	        #sv_InterfaceData.RemotePort := 0;

	    END_IF;

	END_REGION

	REGION 4 – Connection establishment and termination

	    IF (#iqx_Reconnect)                                                     // Reconnect request
	    THEN

	        // Terminate a TCPIP connection if reconnect command available and connection established
	        IF (#sx_Connected)                                                  // Connection established
	        THEN

	            // Disconnect request
	            #sa_Disconnect.Request :=
	            #iqx_Reconnect                                                  // Reconnect command
	            AND #sa_Disconnect.Status = 16#7000;                            // TDISCON block status is equal to 16#7000 (No job processing active)

	            // Terminate a TCPIP connection when request available
	            #sFB_TDISCON(REQ := #sa_Disconnect.Request,
	                         ID := #sv_InterfaceData.ID,
	                         DONE => #sa_Disconnect.Done,
	                         BUSY => #sa_Disconnect.Busy,
	                         ERROR => #sa_Disconnect.Error,
	                         STATUS => #sa_Disconnect.Status);

	            // In case of connection broken, connected bit and disconnect block active bit are reset
	            IF (#sa_Disconnect.Done)                                        // Disconnect was successful
	            THEN

	                #sx_Connected := FALSE;
	                #sa_Disconnect.Active := FALSE;

	                // Connection termination in progress
	            ELSE

	                #sa_Disconnect.Active := TRUE;                              // Set the disconnecting active status bit

	            END_IF;

	            // Try to establish connection if reconnect command active and there is no connection
	        ELSE                                                                // Connection is terminated

	            // Connect request
	            #sa_Connect.Request := #iqx_Reconnect AND                       // Reconnect command
	            #sa_Connect.Status = 16#7000;            // TCON block status is equal to 16#7000 (No job processing active)

	            // Establishing a TCPIP connection when request available
	            #sFB_TCON(REQ := #sa_Connect.Request,
	                      ID := #sv_InterfaceData.ID,
	                      DONE => #sa_Connect.Done,
	                      BUSY => #sa_Connect.Busy,
	                      ERROR => #sa_Connect.Error,
	                      STATUS => #sa_Connect.Status,
	                      CONNECT := #sv_InterfaceData);

	            // In case of connection established, connected bit is set, connect block active bit and reconnect command are reset
	            IF (#sa_Connect.Done)                                           // Connect successful
	            THEN

	                #sx_Connected := TRUE;
	                #sa_Connect.Active := FALSE;
	                #iqx_Reconnect := FALSE;

	                // Connection establishing in progress
	            ELSE

	                #sa_Connect.Active := TRUE;                                 // Set the connecting active status

	            END_IF;

	        END_IF;

	    END_IF;

	END_REGION

	REGION 5 – Connection establishment and termination error handling

	    // Measure the maximum connect or disconnect time
	    #sFB_TimerConTimeout(ix_SignalToDelay := #sa_Connect.Active
	                         OR #sa_Disconnect.Active,
	                         iudi_OnDelayTime := DINT_TO_UDINT(#iUDT_Connection.ConTimeout),
	                         iudi_OffDelayTime := 0);

	    IF (#sFB_TimerConTimeout.qx_DelayedSignal)                                                 // Connecting / disconnecting time error from connection timeout timer
	    THEN

	        IF (#sa_Connect.Active)                                                                  // Connecting is active
	        THEN

	            // If connection already exist and block try establish connection, connected bit is set, connect block active bit and reconnect command are reset
	            IF (#sa_Connect.Status = 16#80A3)                                                    // Connecting status equal to 16#80A3 - The connection already exist
	            THEN

	                #sx_Connected := TRUE;
	                #sa_Connect.Active := FALSE;
	                #iqx_Reconnect := FALSE;

	                // Connection time has expired - error generated
	            ELSE

	                #sx_CommunicationFault := TRUE;

	            END_IF;

	            // Disconnect operation failed - error generated
	        ELSIF (#sa_Disconnect.Active)
	        THEN

	            #sx_CommunicationFault := TRUE;

	        END_IF;

	    END_IF;

	    // The connection terminated by partner - error generated, connected bit reset and reconnect command request set
	    IF (#sa_Diag.Result.State <> 16#04)                         // The connection terminated by partner
	    THEN

	        #sx_CommunicationFault := TRUE;
	        #sx_Connected := FALSE;
	        #iqx_Reconnect := TRUE;

	    END_IF;

	END_REGION

	REGION 6 – Connection diagnostic

	    // Check connection condition ten times per second
	    IF (NOT #sa_Connect.Active AND NOT #sa_Disconnect.Active)        // Connecting and disconnecting procedure are not active
	    THEN

	        #sFB_DIAG(REQ := "DB_Memory".Clock_10Hz,
	                  ID := #sv_InterfaceData.ID,
	                  DONE => #sa_Diag.Done,
	                  BUSY => #sa_Diag.Busy,
	                  ERROR => #sa_Diag.Error,
	                  STATUS => #sa_Diag.Status,
	                  RESULT := #sa_Diag.Result);

	    END_IF;

	END_REGION

	REGION 7 – Connection established filter

	    // Connected status bit filtering
	    #sFB_TimerFilter(ix_SignalToDelay := #sx_Connected,
	                     iudi_OnDelayTime := 50,
	                     qx_DelayedSignal => #sx_ConnectedFiltred);

	END_REGION

	REGION 8 – Statistics

	    // Prepare rising edge of connected status signal
	    #sR_TRIG_ConnectionLost(CLK := NOT #sx_ConnectedFiltred);

	    // Conditions to call "FC_Statistics"
	    IF (NOT #sx_ConnectedFiltred                                                        // No connection
	        OR #iqUDT_EquipmentControl.Command.ResetData)                                  // Reset data
	    THEN

	        "FC_Statistics"(ix_Reset := #iqUDT_EquipmentControl.Command.ResetData,
	                        ix_Activate := NOT #sx_ConnectedFiltred,
	                        ix_RTrigActivate := #sR_TRIG_ConnectionLost.Q,
	                        iqUDT_Statistics := #iqUDT_Statistics.ConnectionLost);

	    END_IF;

	END_REGION

	REGION 9 – Status

	    #sUDT_CommonStatus.Error := #sx_CommunicationFault;                        // Error

	    #sUDT_CommonStatus.AutoON := #sx_ConnectedFiltred;                         // Auto ON

	    #qUDT_HMIStatus.Specific.CommunicationFault := #sx_CommunicationFault;     // Communication faults

	    #qUDT_HMIStatus.Specific.Connected := #sx_ConnectedFiltred;                // Connected

	    IF #sUDT_CommonStatus.AutoON                                               // Auto ON
	    THEN

	        #qUDT_HMIStatus.Status := "DB_HMIStatusConfiguration".AutoON;

	    END_IF;

	    IF #sUDT_CommonStatus.Error                                                // Error
	    THEN

	        #qUDT_HMIStatus.Status := "DB_HMIStatusConfiguration".Error;

	    END_IF;

	END_REGION

	REGION 10 Report to control block

	    // Function to manage report between control block and conveyor block

	    "FC_EquipmentReport"(iUDT_Status := #sUDT_CommonStatus,
	                         iqUDT_Control := #iqUDT_EquipmentControl);

	END_REGION

	REGION 11 – Write outputs

	    #qx_Connected := #sx_Connected;

	END_REGION
END_FUNCTION_BLOCK

TYPE "UDT_ParcelData"
VERSION : 0.1
   STRUCT
      AvgParcelLength : DInt := 10;
      TimeReadMessages : Time := T#10s;
      TimOutComm : Time := T#30s;
      NrOfParcels : Array[1..500] of DInt;
   END_STRUCT;

END_TYPE

TYPE "UDT_UPSSafetyZoneStatistics"
VERSION : 0.1
   STRUCT
      NotHealthy { S7_SetPoint := 'False'} : "UDT_EventStatistic";
   END_STRUCT;

END_TYPE

TYPE "UDT_ConveyorInterface"
TITLE = UDT_ConveyorInterface
VERSION : 0.1
//User-defined structure of conveyor interface variables.
   STRUCT
      Displacement : Int;   // Displacement per PLC scan [cm] either from position (if available) or speed and time
      SpeedSetpoint : Int;   // Conveyor speed setpoint [mm/s]
      ActualSpeed : Int;   // Conveyors actual speed [mm/s]
      DeltaPosition : Int;   // Read from Conveyor Servo Position [mm] after 1 PLC cycle
      RunFwd { ExternalAccessible := 'False'; ExternalVisible := 'False'; ExternalWritable := 'False'} : Bool;   // Run forward request
      RunRvs { ExternalAccessible := 'False'; ExternalVisible := 'False'; ExternalWritable := 'False'} : Bool;   // Run reverse request
      InternalErrorEncoder { ExternalAccessible := 'False'; ExternalVisible := 'False'; ExternalWritable := 'False'} : Bool;   // Encoder has an error
      InternalErrorVFD { ExternalAccessible := 'False'; ExternalVisible := 'False'; ExternalWritable := 'False'} : Bool;   // VFD has an error
      InternalErrorTracking { ExternalAccessible := 'False'; ExternalVisible := 'False'; ExternalWritable := 'False'} : Bool;   // Tracking has an error
      InternalErrorPEC { ExternalAccessible := 'False'; ExternalVisible := 'False'; ExternalWritable := 'False'} : Bool;   // PEC has an error
      InternalWarningVFD { ExternalAccessible := 'False'; ExternalVisible := 'False'; ExternalWritable := 'False'} : Bool;   // VFD has a warning
      InternalWarningTracking { ExternalAccessible := 'False'; ExternalVisible := 'False'; ExternalWritable := 'False'} : Bool;   // Tracking has a warning
      InternalErrorReset { ExternalAccessible := 'False'; ExternalVisible := 'False'; ExternalWritable := 'False'} : Bool;   // Reset internal errors
      ConfigurationError { ExternalAccessible := 'False'; ExternalVisible := 'False'; ExternalWritable := 'False'} : Bool;   // Configuration error is active
      VFDRunning { ExternalAccessible := 'False'; ExternalVisible := 'False'; ExternalWritable := 'False'} : Bool;   // Motor is running
      VFDatSpeed { ExternalAccessible := 'False'; ExternalVisible := 'False'; ExternalWritable := 'False'} : Bool;   // Motor at speed setpoint
      Disconnected { ExternalAccessible := 'False'; ExternalVisible := 'False'; ExternalWritable := 'False'} : Bool;   // VFD disconnected
      ManualModeActive { ExternalAccessible := 'False'; ExternalVisible := 'False'; ExternalWritable := 'False'} : Bool;   // Covneyor is in manual mode
      ResetStatistics { ExternalAccessible := 'False'; ExternalVisible := 'False'; ExternalWritable := 'False'} : Bool;   // Reset statistics
      HardwareOk { ExternalAccessible := 'False'; ExternalVisible := 'False'; ExternalWritable := 'False'} : Bool;   // Hardware for the Equipment is available and healthy
   END_STRUCT;

END_TYPE

FUNCTION_BLOCK "FB_UPSCameraFault"
{ S7_Optimized_Access := 'TRUE' }
VERSION : 0.1
// ATTRIBUTES
// AUTO_NUMBER = True
// BLOCK_NUMBER = 49
// END_ATTRIBUTES
   VAR_INPUT
      ii_GIN { ExternalAccessible := 'False'; ExternalVisible := 'False'; ExternalWritable := 'False'} : Int;   // GIN to be checked
   END_VAR

   VAR_OUTPUT
      qx_Fault { ExternalAccessible := 'False'; ExternalVisible := 'False'; ExternalWritable := 'False'} : Bool;   // Camera fault
   END_VAR

   VAR_IN_OUT
      iqUDT_EquipmentControl : "UDT_EquipmentControl";   // Equipment control structure
   END_VAR

   VAR
      si_CameraGIN { ExternalAccessible := 'False'; ExternalVisible := 'False'; ExternalWritable := 'False'} : Int;   // Camera GIN
      si_MissingScanData { ExternalAccessible := 'False'; ExternalVisible := 'False'; ExternalWritable := 'False'} : Int;   // Number of missing SCAN_DATA2 messages
   END_VAR

   VAR CONSTANT
      ci_MaximumMissingScanData : Int := 10;
   END_VAR


BEGIN
	(*
	----------------------------------------------------------------------------------------

	Version history:
	Date        | Version   | Author        | Remark
	----------------------------------------------------------------------------------------
	15/01/2020  | 3.0       | L.Klar        | 3.0 MHS library release TIA 15.1
	22/02/2023  | 4.0       | F.Baten       | 4.0 Release TIA 17.5
	*)

	REGION 1 - Calculate displacement

	    // Check if for GIN found in tracking ID has been created (SCAN_DATA2 received)
	    // After 10 missings a fault is generated

	    IF #ii_GIN <> #si_CameraGIN
	        AND #ii_GIN <> 0
	    THEN

	        #si_CameraGIN := #ii_GIN;

	        IF #si_CameraGIN > 0
	        THEN
	            IF NOT "DB_GIN".GIN[#si_CameraGIN].UPS.IDCreated
	            THEN
	                #si_MissingScanData += 1;
	            ELSE
	                #si_MissingScanData := 0;
	            END_IF;
	        END_IF;


	        IF #si_MissingScanData >= #ci_MaximumMissingScanData
	        THEN
	            #qx_Fault := TRUE;
	        END_IF;

	    END_IF;

	END_REGION

	REGION 2 - Fault reset
	    IF #si_MissingScanData >= #ci_MaximumMissingScanData
	        AND #iqUDT_EquipmentControl.Command.Reset
	    THEN
	        #qx_Fault := FALSE;
	        #si_MissingScanData := 0;
	    END_IF;
	END_REGION
END_FUNCTION_BLOCK

FUNCTION_BLOCK "FB_UPSCIP"
TITLE = Communication Interface Panel Cabinet Block
{ S7_Optimized_Access := 'TRUE' }
AUTHOR : CesarLeite
VERSION : 0.1
// ATTRIBUTES
// AUTO_NUMBER = True
// BLOCK_NUMBER = 51
// END_ATTRIBUTES
   VAR_INPUT
      ix_SystemRunning { ExternalAccessible := 'False'; ExternalVisible := 'False'; ExternalWritable := 'False'} : Bool;   // System running error free
      ix_XLESelectorSwitch { ExternalAccessible := 'False'; ExternalVisible := 'False'; ExternalWritable := 'False'} : Bool;   // Selector switch CHAT/XLE - (True=BackUp, False=Primary)
      ix_CameraSelectorSwitch { ExternalAccessible := 'False'; ExternalVisible := 'False'; ExternalWritable := 'False'} : Bool;   // Selector switch Camera - (True=BackUp, False=Primary)
      ix_CIP24VDC { ExternalAccessible := 'False'; ExternalVisible := 'False'; ExternalWritable := 'False'} : Bool;   // CIP 24VDC Ok - (True=Healthy, False=Error)
      ix_CIPCircuitBreakerOk { ExternalAccessible := 'False'; ExternalVisible := 'False'; ExternalWritable := 'False'} : Bool;   // CIP circuit breaker Ok (True=Healthy, False=Error)
      ix_DWSOk { ExternalAccessible := 'False'; ExternalVisible := 'False'; ExternalWritable := 'False'} : Bool;   // Weighing Scale Ok (True=Healthy, False=Error)
      ix_CameraInput1 { ExternalAccessible := 'False'; ExternalVisible := 'False'; ExternalWritable := 'False'} : Bool;   // Camera Tunel Input 1
      ix_CameraInput2 { ExternalAccessible := 'False'; ExternalVisible := 'False'; ExternalWritable := 'False'} : Bool;   // Camera Tunel Input 2
      ix_XLEFaulty { ExternalAccessible := 'False'; ExternalVisible := 'False'; ExternalWritable := 'False'} : Bool;   // XLE Chat communication fault
   END_VAR

   VAR_OUTPUT
      qUDT_HMIStatus { ExternalAccessible := 'False'; ExternalVisible := 'False'; ExternalWritable := 'False'} : "UDT_UPSCIPStatus";   // CIP Status
      qUDT_Status { ExternalAccessible := 'False'; ExternalVisible := 'False'; ExternalWritable := 'False'} : "UDT_CommonStatus";   // CIP HMI Status
      qx_SystemStopRequest { ExternalAccessible := 'False'; ExternalVisible := 'False'; ExternalWritable := 'False'} : Bool;   // System stop request
      qx_XLEReconnect { ExternalAccessible := 'False'; ExternalVisible := 'False'; ExternalWritable := 'False'} : Bool;   // Reconnect XLE
      qx_XLESwitch { ExternalAccessible := 'False'; ExternalVisible := 'False'; ExternalWritable := 'False'} : Bool;   // If the output is false the XLE is in primary, if false the XLE is in backup
      qx_CameraSwitch { ExternalAccessible := 'False'; ExternalVisible := 'False'; ExternalWritable := 'False'} : Bool;   // If the output is false the camera is in primary, if false the camara is in backup
   END_VAR

   VAR_IN_OUT
      iqUDT_EquipmentControl : "UDT_EquipmentControl";   // CIP Equipment control
      iqUDT_Statistics : "UDT_UPSCIPStatistics";   // CIP Statistics structure
   END_VAR

   VAR
      sUDT_HMIStatus { ExternalAccessible := 'False'; ExternalVisible := 'False'; ExternalWritable := 'False'; S7_SetPoint := 'False'} : "UDT_UPSCIPStatus";   // HMI status structure
      sUDT_CommonStatus { ExternalAccessible := 'False'; ExternalVisible := 'False'; ExternalWritable := 'False'; S7_SetPoint := 'False'} : "UDT_CommonStatus";   // Common status structure
      sUDT_CommonStatusOld { ExternalAccessible := 'False'; ExternalVisible := 'False'; ExternalWritable := 'False'; S7_SetPoint := 'False'} : "UDT_CommonStatus";   // Common status structure
      sR_Trig_XLESwitch {InstructionName := 'R_TRIG'; LibVersion := '1.0'; ExternalAccessible := 'False'; ExternalVisible := 'False'; ExternalWritable := 'False'; S7_SetPoint := 'False'} : R_TRIG;   // Rise trigger when XLE selector switch to backup
      sF_Trig_XLESwitch {InstructionName := 'F_TRIG'; LibVersion := '1.0'; ExternalAccessible := 'False'; ExternalVisible := 'False'; ExternalWritable := 'False'; S7_SetPoint := 'False'} : F_TRIG;   // Fall trigger when XLE selector switch to primary
      sR_Trig_CameraSwitch {InstructionName := 'R_TRIG'; LibVersion := '1.0'; ExternalAccessible := 'False'; ExternalVisible := 'False'; ExternalWritable := 'False'; S7_SetPoint := 'False'} : R_TRIG;   // Rise trigger when camera selector switch to backup
      sF_Trig_CameraSwitch {InstructionName := 'F_TRIG'; LibVersion := '1.0'; ExternalAccessible := 'False'; ExternalVisible := 'False'; ExternalWritable := 'False'; S7_SetPoint := 'False'} : F_TRIG;   // Fall trigger when camera selector switch to primary
      sF_Trig_CIP24VDC {InstructionName := 'F_TRIG'; LibVersion := '1.0'; ExternalAccessible := 'False'; ExternalVisible := 'False'; ExternalWritable := 'False'; S7_SetPoint := 'False'} : F_TRIG;   // Fall trigger when CIP 24VDC
      sF_Trig_CIPCircuitBreaker {InstructionName := 'F_TRIG'; LibVersion := '1.0'; ExternalAccessible := 'False'; ExternalVisible := 'False'; ExternalWritable := 'False'; S7_SetPoint := 'False'} : F_TRIG;   // Fall trigger when CIP circuit breaker is tripped
      sF_Trig_DWSFault {InstructionName := 'F_TRIG'; LibVersion := '1.0'; ExternalAccessible := 'False'; ExternalVisible := 'False'; ExternalWritable := 'False'; S7_SetPoint := 'False'} : F_TRIG;   // Fall trigger when weighing scale has a fault
   END_VAR


BEGIN
	(*
	----------------------------------------------------------------------------------------

	Version history:
	Date        | Version   | Author        | Remark
	----------------------------------------------------------------------------------------
	19/09/2019  | 2.0       | C.Leite       | first release TIA 15.1
	14/10/2019  | 2.1       | L.Klar        | Updated status structure
	07/11/2019  | 2.2       | M.Kurc        | Add I/O: system running/stop and camera/XLE switch
	12/11/2019  | 3.0       | P.Majka       | 3.0 MHS library release TIA 15.1
	09/07/2020  | 3.1       | S.Theocharis  | Update HMI status in every scan. Bug fix with initialization
	21/08/2020  | 3.2       | S.Theocharis  | Error handling when XLE/Camera switch while system is running
	                                        | Added statistics of selection switches
	13/08/2020  | 3.3       | L.Klar        | XLE reconnect command added, communication fault added to stop camera belt
	22/02/2023  | 4.0       | F.Baten       | 4.0 Release TIA 17.5
	*)

	REGION 1 - Trigger

	    // Rise trigger selector switch CHAT/XLE BackUp
	    #sR_Trig_XLESwitch(CLK := #ix_XLESelectorSwitch);

	    // Fall trigger selector switch CHAT/XLE BackUp
	    #sF_Trig_XLESwitch(CLK := #ix_XLESelectorSwitch);

	    // Fall trigger selector switch camera to primary
	    #sF_Trig_CameraSwitch(CLK := #ix_CameraSelectorSwitch);

	    // Rise trigger selector switch camera to primary
	    #sR_Trig_CameraSwitch(CLK := #ix_CameraSelectorSwitch);

	    // Fall trigger CIP 24VDC error
	    #sF_Trig_CIP24VDC(CLK := #ix_CIP24VDC);

	    // Fall trigger CIP 24VDC circuit breaker tripped
	    #sF_Trig_CIPCircuitBreaker(CLK := #ix_CIPCircuitBreakerOk);

	    // Fall trigger weighing scale fault
	    #sF_Trig_DWSFault(CLK := #ix_DWSOk);

	END_REGION

	REGION 2 - Reset faults

	    // All faults are reset when the reset input is true
	    IF #iqUDT_EquipmentControl.Command.Reset
	    THEN

	        #sUDT_HMIStatus.Specific.CIP24VDCError := FALSE;
	        #sUDT_HMIStatus.Specific.CIPCircuitBreakerTripped := FALSE;
	        #sUDT_HMIStatus.Specific.WeighingScaleFault := FALSE;
	        #sUDT_HMIStatus.Specific.XLE_SwitchError := FALSE;
	        #sUDT_HMIStatus.Specific.Camera_SwitchError := FALSE;
	    END_IF;

	END_REGION

	REGION 3 - Status monitoring

	    // CHAT/XLE Selector Switch

	    #sUDT_HMIStatus.Specific.XLEBackUp := #ix_XLESelectorSwitch;

	    #sUDT_HMIStatus.Specific.XLEPrimary := NOT #ix_XLESelectorSwitch;

	    // CIP 24VDC Fault

	    IF NOT #ix_CIP24VDC
	    THEN

	        #sUDT_HMIStatus.Specific.CIP24VDCError := TRUE;

	    END_IF;

	    // CIP Circuit Breaker Tripped

	    IF NOT #ix_CIPCircuitBreakerOk
	    THEN

	        #sUDT_HMIStatus.Specific.CIPCircuitBreakerTripped := TRUE;

	    END_IF;

	    // Weighing Scale Fault

	    IF NOT #ix_DWSOk
	    THEN

	        #sUDT_HMIStatus.Specific.WeighingScaleFault := TRUE;

	    END_IF;

	    // Camera Tunel
	    #sUDT_HMIStatus.Specific.CameraTunel1 := NOT #ix_CameraSelectorSwitch;
	    #sUDT_HMIStatus.Specific.CameraTunel2 := #ix_CameraSelectorSwitch;

	    // XLE Switching error while running
	    IF #ix_SystemRunning AND (#sR_Trig_XLESwitch.Q OR #sF_Trig_XLESwitch.Q)
	    THEN
	        #sUDT_HMIStatus.Specific.XLE_SwitchError := TRUE;
	    END_IF;

	    // Camera Switching error while running
	    IF #ix_SystemRunning AND (#sR_Trig_CameraSwitch.Q OR #sF_Trig_CameraSwitch.Q)
	    THEN
	        #sUDT_HMIStatus.Specific.Camera_SwitchError := TRUE;
	    END_IF;

	END_REGION

	REGION 4 - Switching Camera and XLE

	    // XLE activation
	    #qx_XLESwitch := #ix_XLESelectorSwitch;

	    // Camera activation
	    #qx_CameraSwitch := #ix_CameraSelectorSwitch;

	END_REGION

	REGION 5 - XLE change

	    #qx_XLEReconnect := #sR_Trig_XLESwitch.Q OR #sF_Trig_XLESwitch.Q;

	END_REGION

	REGION 6 - Statistics

	    // 24 VDC fault statistics
	    IF #sUDT_HMIStatus.Specific.CIP24VDCError
	        OR #iqUDT_EquipmentControl.Command.ResetData
	    THEN

	        "FC_Statistics"(ix_Reset := #iqUDT_EquipmentControl.Command.ResetData,
	                        ix_Activate := #sUDT_HMIStatus.Specific.CIP24VDCError,
	                        ix_RTrigActivate := #sF_Trig_CIP24VDC.Q,
	                        iqUDT_Statistics := #iqUDT_Statistics.CIP24VDCFault);

	    END_IF;

	    // CIP Circuit Breaker Tripped statistics
	    IF #sUDT_HMIStatus.Specific.CIPCircuitBreakerTripped
	        OR #iqUDT_EquipmentControl.Command.ResetData
	    THEN

	        "FC_Statistics"(ix_Reset := #iqUDT_EquipmentControl.Command.ResetData,
	                        ix_Activate := #sUDT_HMIStatus.Specific.CIPCircuitBreakerTripped,
	                        ix_RTrigActivate := #sF_Trig_CIPCircuitBreaker.Q,
	                        iqUDT_Statistics := #iqUDT_Statistics.CIPCircuitBreakerTripped);

	    END_IF;

	    // CIP Weighing Scale Fault statistics
	    IF #sUDT_HMIStatus.Specific.WeighingScaleFault
	        OR #iqUDT_EquipmentControl.Command.ResetData
	    THEN

	        "FC_Statistics"(ix_Reset := #iqUDT_EquipmentControl.Command.ResetData,
	                        ix_Activate := #sUDT_HMIStatus.Specific.WeighingScaleFault,
	                        ix_RTrigActivate := #sF_Trig_DWSFault.Q,
	                        iqUDT_Statistics := #iqUDT_Statistics.WeighingScaleFault);
	    END_IF;

	    //Camera selection switch changes
	    IF #sR_Trig_CameraSwitch.Q OR #sF_Trig_CameraSwitch.Q THEN
	        #iqUDT_Statistics.SS_Camera += 1;

	    ELSIF #iqUDT_EquipmentControl.Command.ResetData THEN
	        #iqUDT_Statistics.SS_Camera := 0;
	    END_IF;

	    //XLE selector switch changes
	    IF #sR_Trig_XLESwitch.Q OR #sF_Trig_XLESwitch.Q THEN
	        #iqUDT_Statistics.SS_XLE += 1;

	    ELSIF #iqUDT_EquipmentControl.Command.ResetData THEN
	        #iqUDT_Statistics.SS_XLE := 0;
	    END_IF;

	END_REGION

	REGION 7 - Status

	    // Stop system
	    #qx_SystemStopRequest := #ix_SystemRunning AND (#sUDT_HMIStatus.Specific.Camera_SwitchError OR #sUDT_HMIStatus.Specific.XLE_SwitchError OR #ix_XLEFaulty);

	    // Set common error to report
	    #sUDT_CommonStatus.Error := #sUDT_HMIStatus.Specific.WeighingScaleFault
	    OR #sUDT_HMIStatus.Specific.CIPCircuitBreakerTripped
	    OR #sUDT_HMIStatus.Specific.CIP24VDCError
	    OR #sUDT_HMIStatus.Specific.Camera_SwitchError
	    OR #sUDT_HMIStatus.Specific.XLE_SwitchError;

	    // Write status value to output
	    IF #sUDT_CommonStatusOld <> #sUDT_CommonStatus                                // Update on change
	        OR (#sR_Trig_CameraSwitch.Q OR #sF_Trig_CameraSwitch.Q)
	        OR (#sR_Trig_XLESwitch.Q OR #sF_Trig_XLESwitch.Q)
	    THEN

	        #sUDT_HMIStatus.Status := 0; //initialize status

	        IF #sUDT_HMIStatus.Specific.WeighingScaleFault                             // Error
	            OR #sUDT_HMIStatus.Specific.Camera_SwitchError
	            OR #sUDT_HMIStatus.Specific.XLE_SwitchError
	        THEN

	            #sUDT_HMIStatus.Status := "DB_HMIStatusConfiguration".Error;

	        END_IF;

	        IF #sUDT_HMIStatus.Specific.CIPCircuitBreakerTripped                       // CB error
	            OR #sUDT_HMIStatus.Specific.CIP24VDCError
	        THEN

	            #sUDT_HMIStatus.Status := "DB_HMIStatusConfiguration".CBError;
	        END_IF;


	        #sUDT_CommonStatusOld := #sUDT_CommonStatus;                              // Copy status to memory
	        #qUDT_Status := #sUDT_CommonStatus;                                       // Copy status to output
	    END_IF;

	    #qUDT_HMIStatus := #sUDT_HMIStatus;                                           // Copy HMI status

	END_REGION

	REGION 8 - Report to control block

	    // Function to manage report between control block and conveyor block

	    "FC_EquipmentReport"(iUDT_Status := #sUDT_CommonStatus,
	                         iqUDT_Control := #iqUDT_EquipmentControl);

	END_REGION

END_FUNCTION_BLOCK

FUNCTION_BLOCK "FB_SickTCPcomm"
{ S7_Optimized_Access := 'TRUE' }
VERSION : 0.1
// ATTRIBUTES
// AUTO_NUMBER = True
// BLOCK_NUMBER = 236
// END_ATTRIBUTES
   VAR_INPUT
      i_UDT_Connection { ExternalAccessible := 'False'; ExternalVisible := 'False'; ExternalWritable := 'False'} : "UDT_Connection";   // Connection parameters
   END_VAR

   VAR_OUTPUT
      qx_CommunicationError { ExternalAccessible := 'False'; ExternalVisible := 'False'; ExternalWritable := 'False'} : Bool;   // Communication error
      q_di_FlowCount { ExternalAccessible := 'False'; ExternalVisible := 'False'; ExternalWritable := 'False'} : DInt;   // Total parcel flow count
   END_VAR

   VAR_IN_OUT
      iq_UDT_EquipmentControl : "UDT_EquipmentControl";   // Equipment control structure
      iq_UDT_Statistics_Connect : "UDT_TCPIPConnectStatistics";   // Statistic structure
      iq_UDT_Statistics_Rcv : "UDT_TCPIPReceiveStatistics";   // Statistic structure
      iq_UDT_ParcelData : "UDT_ParcelData";   // Parcel data
      iq_UDT_FIFOHeader : "UDT_FifoHeader";
      iq_FIFOData : Array[*] of "UDT_Message";
      iqx_Reconnect { ExternalAccessible := 'False'; ExternalVisible := 'False'; ExternalWritable := 'False'} : Bool;   // Reconnect command
   END_VAR

   VAR
      TCPIP_Connect { ExternalAccessible := 'False'; ExternalVisible := 'False'; ExternalWritable := 'False'; S7_SetPoint := 'False'} : "FB_TCPIPConnect";
      TCPIPReceive { ExternalAccessible := 'False'; ExternalVisible := 'False'; ExternalWritable := 'False'; S7_SetPoint := 'False'} : "FB_SickVmsTcpipReceive";
      ss_Status { ExternalAccessible := 'False'; ExternalVisible := 'False'; ExternalWritable := 'False'} : Struct   // Status structure
         ErrorCode { ExternalAccessible := 'False'; ExternalVisible := 'False'; ExternalWritable := 'False'} : Struct   // Error code structure
            TRCV { ExternalAccessible := 'False'; ExternalVisible := 'False'; ExternalWritable := 'False'} : Word;   // Siemens TRCV error code - Check documentation
         END_STRUCT;
         FIFORcvStatus { ExternalAccessible := 'False'; ExternalVisible := 'False'; ExternalWritable := 'False'} : "UDT_FifoStatus";   // Receive FIFO status structure
         FIFORcvError { ExternalAccessible := 'False'; ExternalVisible := 'False'; ExternalWritable := 'False'; S7_SetPoint := 'True'} : Bool;   // Receive FIFO error
         FIFORcvWarning { ExternalAccessible := 'False'; ExternalVisible := 'False'; ExternalWritable := 'False'; S7_SetPoint := 'True'} : Bool;   // Receive  FIFO warning
         ReceiveError { ExternalAccessible := 'False'; ExternalVisible := 'False'; ExternalWritable := 'False'} : Bool;   // TRCV block operation error - Check TRCVStatus
      END_STRUCT;
      ss_UDT_MsgArray { ExternalAccessible := 'False'; ExternalVisible := 'False'; ExternalWritable := 'False'; S7_SetPoint := 'False'} : "UDT_Message";   // Message character array
      sdi_Lenght { ExternalAccessible := 'False'; ExternalVisible := 'False'; ExternalWritable := 'False'} : DInt;   // object length
      si_SystemStatus { ExternalAccessible := 'False'; ExternalVisible := 'False'; ExternalWritable := 'False'} : Int;   // 0=stopped, 1=running, 2=jam
      si_PackageCount { ExternalAccessible := 'False'; ExternalVisible := 'False'; ExternalWritable := 'False'} : Int;   // number of objects
      si_SeqNr { ExternalAccessible := 'False'; ExternalVisible := 'False'; ExternalWritable := 'False'} : Int;   // Current incremental sequence number
      si_SeqNrOld { ExternalAccessible := 'False'; ExternalVisible := 'False'; ExternalWritable := 'False'} : Int;   // Last incremental sequence number
      si_Counter { ExternalAccessible := 'False'; ExternalVisible := 'False'; ExternalWritable := 'False'} : Int;   // loop counter
      slr_Time { ExternalAccessible := 'False'; ExternalVisible := 'False'; ExternalWritable := 'False'} : LReal;   // message read time
      slr_ComTimeOut { ExternalAccessible := 'False'; ExternalVisible := 'False'; ExternalWritable := 'False'} : LReal;   // Communcation timeout time
      sx_CommError { ExternalAccessible := 'False'; ExternalVisible := 'False'; ExternalWritable := 'False'} : Bool;   // Communication error
      sx_ReceiveEnable { ExternalAccessible := 'False'; ExternalVisible := 'False'; ExternalWritable := 'False'} : Bool;   // TRUE=receive enable
      sx_ReadBuffer { ExternalAccessible := 'False'; ExternalVisible := 'False'; ExternalWritable := 'False'} : Bool;   // read the FIFO buffer
      sr_TotalAvgParcel { ExternalAccessible := 'False'; ExternalVisible := 'False'; ExternalWritable := 'False'} : Real;
   END_VAR

   VAR_TEMP
      tx_Error : Bool;   // TCPIP communication error
      tdi_CycleLenght : DInt;
      tx_Warning : Bool;   // TCPIP communication warning
      ti_Length : Int;   // the length of parcel
      ti_Move_BLKErrorCode : Int;
      tr_CycleAvgParcels : Real;
      tx_IntegerAvgParcels : Real;
   END_VAR

   VAR CONSTANT
      Index_IncSeqNr : Int := 1;   // was 8
      Index_SystemStatus : Int := 5;   // was 12
      Index_PackageCount : Int := 6;   // was 13
      Index_StartFirstLength : Int := 7;   // was 14
   END_VAR


BEGIN
	(*
	----------------------------------------------------------------------------------------
	|                                                                                      |
	|  Copyright  2019             MHS                                                     |
	|  All Rights Reserved         Larenweg 90                                             |
	|                              5234 KC 's-Hertogenbosch,                               |
	|                              Netherlands                                             |
	|                                                                                      |
	----------------------------------------------------------------------------------------

	Version history:
	Date        | Version   | Author       | Remark
	----------------------------------------------------------------------------------------
	22/03/2021  | 0.1       | M. Jager     | first release MHS TIA 16.0
	26/07/2022  | 0.2       | S. Deulkar   | Reset avg parcel data when reset data command occour
	14/03/2024  | 4.1       | S. Nieswiec  | Added from Hannover project and changed name according to standard
	*)


	#TCPIP_Connect(iUDT_Connection := #i_UDT_Connection,
	               qx_Connected => #sx_ReceiveEnable,
	               iqUDT_EquipmentControl := #iq_UDT_EquipmentControl,
	               iqUDT_Statistics := #iq_UDT_Statistics_Connect,
	               iqx_Reconnect := #iqx_Reconnect);

	#TCPIPReceive(i_UDT_Connection := #i_UDT_Connection,
	              ix_EnableReceive := #sx_ReceiveEnable,
	              qx_Error => #tx_Error,
	              qx_Warning => #tx_Warning,
	              iq_UDT_FifoHeader := #iq_UDT_FIFOHeader,
	              iqs_FifoData := #iq_FIFOData,
	              iq_UDT_Statistics := #iq_UDT_Statistics_Rcv);


	// Read the FIFO data when it is not EMPTY
	IF NOT #iq_UDT_FIFOHeader.Status.Empty THEN
	    #sx_ReadBuffer := TRUE;
	END_IF;

	IF #sx_ReadBuffer THEN

	    "FC_Fifo"(ic_Mode := 'R',
	              qUDT_Status => #ss_Status.FIFORcvStatus,
	              qx_Error => #ss_Status.FIFORcvError,
	              qx_Warning => #ss_Status.FIFORcvWarning,
	              iqv_Data := #ss_UDT_MsgArray,
	              iqUDT_FifoHeader := #iq_UDT_FIFOHeader,
	              iqv_DataBuffer := #iq_FIFOData);

	    #sx_ReadBuffer := FALSE;

	    //System status
	    #si_SystemStatus := (STRING_TO_INT(IN := (CHAR_TO_STRING(IN := #ss_UDT_MsgArray.Character[#Index_SystemStatus]))));

	    //Package count
	    #si_PackageCount := (STRING_TO_INT(IN := (CHAR_TO_STRING(IN := #ss_UDT_MsgArray.Character[#Index_PackageCount]))));

	    #tdi_CycleLenght := 0;

	    FOR #si_Counter := 1 TO #si_PackageCount BY 1 DO
	        //get length from FIFO data and add to total length

	        "FC_CharToInt"(Offset := (#Index_StartFirstLength + ((#si_Counter - 1) * 12)),
	                       Data := #ss_UDT_MsgArray,
	                       qi_data => #ti_Length);

	        #sdi_Lenght := #sdi_Lenght + #ti_Length;

	        #tdi_CycleLenght += #ti_Length;

	    END_FOR;

	    IF #iq_UDT_EquipmentControl.Command.ResetData
	    THEN
	        #sr_TotalAvgParcel := 0;
	    END_IF;

	    #tr_CycleAvgParcels := (DINT_TO_REAL(#tdi_CycleLenght) / DINT_TO_REAL(#iq_UDT_ParcelData.AvgParcelLength));

	    #sr_TotalAvgParcel += #tr_CycleAvgParcels;

	    IF #sr_TotalAvgParcel < 0
	    THEN
	        #sr_TotalAvgParcel := 0;
	    END_IF;

	    //get incremental sequence number
	    "FC_CharToInt"(Offset := #Index_IncSeqNr,
	                   Data := #ss_UDT_MsgArray,
	                   qi_data => #si_SeqNr);

	    // when incremental sequence number changed, reset timer communication error
	    IF #si_SeqNr <> #si_SeqNrOld THEN
	        #slr_ComTimeOut := 0;
	        #sx_CommError := FALSE;
	        #si_SeqNrOld := #si_SeqNr;
	    END_IF;

	END_IF;

	// Output flow count
	#q_di_FlowCount := TRUNC(#sr_TotalAvgParcel);

	//If time elapsed, store  NrOfParcelsinto DB_ParcelData
	#slr_Time := #slr_Time + "DB_Memory".PrevCycleTime;
	IF (#slr_Time > LINT_TO_REAL(IN := TIME_TO_LINT(IN := #iq_UDT_ParcelData.TimeReadMessages))) THEN

	    // Shift Parcel data with 1 position
	    MOVE_BLK(IN := #iq_UDT_ParcelData.NrOfParcels[1],
	             COUNT := 499,
	             OUT => #iq_UDT_ParcelData.NrOfParcels[2]);

	    //calculate number of parcels and store in DB_ParcelData
	    #iq_UDT_ParcelData.NrOfParcels[1] := #sdi_Lenght / #iq_UDT_ParcelData.AvgParcelLength;

	    //reset time and length
	    #slr_Time := 0.0;
	    #sdi_Lenght := 0;
	END_IF;

	//TimeOut Communication
	#slr_ComTimeOut := #slr_ComTimeOut + "DB_Memory".PrevCycleTime;
	IF (#slr_ComTimeOut > LINT_TO_REAL(IN := TIME_TO_LINT(IN := #iq_UDT_ParcelData.TimOutComm))) THEN
	    #sx_CommError := TRUE;
	    #slr_ComTimeOut := 0;
	END_IF;


	//Write Error Status
	#iq_UDT_EquipmentControl.Report.Error := #iq_UDT_EquipmentControl.Report.Error OR #sx_CommError;
	#qx_CommunicationError := #sx_CommError;
END_FUNCTION_BLOCK

FUNCTION_BLOCK "FB_UPS2ndStageFlowControl"
{ S7_Optimized_Access := 'TRUE' }
VERSION : 0.1
// ATTRIBUTES
// AUTO_NUMBER = True
// BLOCK_NUMBER = 47
// END_ATTRIBUTES
   VAR_INPUT
      ix_LengthBased { ExternalAccessible := 'False'; ExternalVisible := 'False'; ExternalWritable := 'False'} : Bool;
      ix_ImperialLength { ExternalAccessible := 'False'; ExternalVisible := 'False'; ExternalWritable := 'False'} : Bool;
      ix_IncrementingCounts { ExternalAccessible := 'False'; ExternalVisible := 'False'; ExternalWritable := 'False'} : Bool;
      idi_ParcelCountInfeed { ExternalAccessible := 'False'; ExternalVisible := 'False'; ExternalWritable := 'False'} : DInt;   //  Counter of parcels from infeed
      ix_ActiveInfeed { ExternalAccessible := 'False'; ExternalVisible := 'False'; ExternalWritable := 'False'} : Bool;   //  Infeed is running / active
   END_VAR

   VAR_OUTPUT
      qx_New15SecInterval { ExternalAccessible := 'False'; ExternalVisible := 'False'; ExternalWritable := 'False'} : Bool;   //  TRUE = Indicates a new 15 Sec interval to partner PLC
      qx_LimitFlowInfeed { ExternalAccessible := 'False'; ExternalVisible := 'False'; ExternalWritable := 'False'} : Bool;   //  TRUE = Stop infeed due flow control
      qdi_30secFlowInfeed { ExternalAccessible := 'False'; ExternalVisible := 'False'; ExternalWritable := 'False'} : DInt;   //  30 seconds pph rate
      qdi_1minFlowInfeed { ExternalAccessible := 'False'; ExternalVisible := 'False'; ExternalWritable := 'False'} : DInt;   //  1 minute pph rate
      qdi_3minFlowInfeed { ExternalAccessible := 'False'; ExternalVisible := 'False'; ExternalWritable := 'False'} : DInt;   //  3 minutes pph rate
      qdi_10minFlowInfeed { ExternalAccessible := 'False'; ExternalVisible := 'False'; ExternalWritable := 'False'} : DInt;   //  10 minutes pph rate
   END_VAR

   VAR_IN_OUT
      iqUDT_EquipmentControl : "UDT_EquipmentControl";
      iq_InfeedArray : "UDT_UPSFlowRateCountingRegisters";   //  Array of line x
      iqUDT_FlowControlHMI : "UDT_UPSFlowControlHMI";
   END_VAR

   VAR
      s_FB_Pulse_EndOf15sPeriod { ExternalAccessible := 'False'; ExternalVisible := 'False'; ExternalWritable := 'False'; S7_SetPoint := 'False'} : "FB_Pulse";   //  15 second pulse generator
      s_infeed { ExternalAccessible := 'False'; ExternalVisible := 'False'; ExternalWritable := 'False'} : Struct   //  Data of infeed line
         diCounter { ExternalAccessible := 'False'; ExternalVisible := 'False'; ExternalWritable := 'False'} : DInt;   //  Counter of parcels from infeed
         diLastScanCounter { ExternalAccessible := 'False'; ExternalVisible := 'False'; ExternalWritable := 'False'} : DInt;   //  Last scan counter of parcels from infeed
         diFlowRate30sec { ExternalAccessible := 'False'; ExternalVisible := 'False'; ExternalWritable := 'False'} : DInt;   //  30sec pph rate
         diFlowRate1min { ExternalAccessible := 'False'; ExternalVisible := 'False'; ExternalWritable := 'False'} : DInt;   //  1 min pph rate
         diFlowRate3min { ExternalAccessible := 'False'; ExternalVisible := 'False'; ExternalWritable := 'False'} : DInt;   //  3 min pph rate
         diFlowRate10min { ExternalAccessible := 'False'; ExternalVisible := 'False'; ExternalWritable := 'False'} : DInt;   //  10 min pph rate
         iNumberOfNewParcels { ExternalAccessible := 'False'; ExternalVisible := 'False'; ExternalWritable := 'False'} : Int;   //  Number of new parcels during this scan
         Active { ExternalAccessible := 'False'; ExternalVisible := 'False'; ExternalWritable := 'False'} : Bool;   //  TRUE = infeed is active
         RequestStop { ExternalAccessible := 'False'; ExternalVisible := 'False'; ExternalWritable := 'False'} : Bool;   //  TRUE= Request flow control
         OneShotRequestStop { ExternalAccessible := 'False'; ExternalVisible := 'False'; ExternalWritable := 'False'} : Bool;   //  Rising edge request to stop
         DuringMinimumStopTime { ExternalAccessible := 'False'; ExternalVisible := 'False'; ExternalWritable := 'False'} : Bool;   //  Infeed is stopped and the minimum stop time is not elapsed
      END_STRUCT;
      s_FB_MinStopTimeActive { ExternalAccessible := 'False'; ExternalVisible := 'False'; ExternalWritable := 'False'; S7_SetPoint := 'False'} : "FB_TimerOnOffDelay";   //  Minimum stop time active
      sx_Disabled { ExternalAccessible := 'False'; ExternalVisible := 'False'; ExternalWritable := 'False'} : Bool;   // Disabled from user
      sdi_CumulativeFlowRate { ExternalAccessible := 'False'; ExternalVisible := 'False'; ExternalWritable := 'False'} : DInt;   //  Cumulative flow rate 1min pph at evaluation point
      sdi_AverageLength { ExternalAccessible := 'False'; ExternalVisible := 'False'; ExternalWritable := 'False'} : DInt;   //  Average length
      si_LastLowPriority { ExternalAccessible := 'False'; ExternalVisible := 'False'; ExternalWritable := 'False'} : Int;   //  Pointer to the last low priority infeed
      si_limit { ExternalAccessible := 'False'; ExternalVisible := 'False'; ExternalWritable := 'False'} : Int;   //  Number of infeeds in use - uper limit for array
      si_CurrentConsecutivesAboveSP { ExternalAccessible := 'False'; ExternalVisible := 'False'; ExternalWritable := 'False'} : Int;   //  Number of consecutive intervals  with flow above HMI set point
      si_CurrentConsecutivesBelowSP { ExternalAccessible := 'False'; ExternalVisible := 'False'; ExternalWritable := 'False'} : Int;   //  Number of consecutive intervals with flow below HMI set point
      sx_StopRequested { ExternalAccessible := 'False'; ExternalVisible := 'False'; ExternalWritable := 'False'} : Bool;   //  Any infeed requested to stop
   END_VAR

   VAR_TEMP
      tr_quotient : Real;   //  Quotient of division
      tr_fraction : Real;   //  Return of fraction
      ti_buffer : Int;   //  Auxiliary buffer
      ti_LC_k : Int;
      ti_Index : Int;   //  temporaty index
      tx_End15sPeriod : Bool;   //  End of 15 seconds flow period
   END_VAR

   VAR CONSTANT
      cdi_InchesAverageLength : DInt := DINT#20;   //  Average length in inches
      cdi_mmAverageLength : DInt := DINT#508;   //  Average length in mm
   END_VAR


BEGIN
	(*
	----------------------------------------------------------------------------------------
	|                                                                                      |
	|  Copyright  2019             MHS                                                     |
	|  All Rights Reserved         Larenweg 90                                             |
	|                              5234 KC 's-Hertogenbosch,                               |
	|                              Netherlands                                             |
	|                                                                                      |
	----------------------------------------------------------------------------------------

	Version history:
	Date        | Version   | Author       | Remark
	----------------------------------------------------------------------------------------
	28/01/2020  | 3.0       | S.Theocharis | Initial version (Covnert from 1st stage)
	14/03/2024  | 4.1       | S.Nieswiec   | Added from Hannover project
	*)

	REGION 1 - Normalization and data move

	    REGION 1.1 - Normalization

	        IF #ix_LengthBased THEN

	            IF #ix_ImperialLength THEN
	                #sdi_AverageLength := #cdi_InchesAverageLength;  // infeed count in inches
	            ELSE
	                #sdi_AverageLength := #cdi_mmAverageLength;       // infeed count in mm
	            END_IF;
	        ELSE
	            #sdi_AverageLength := L#1;                            // infeed count in parcels
	        END_IF;

	    END_REGION

	    REGION 1.2 - Move Input data to static
	        //Move counters
	        #s_infeed.diCounter := #idi_ParcelCountInfeed;


	        //Move infeed active bit
	        #s_infeed.Active := #ix_ActiveInfeed;


	    END_REGION

	END_REGION


	REGION 2 - End of 15s flow period

	    // Calculate 15 seconds period
	    #s_FB_Pulse_EndOf15sPeriod(iudi_PulseTime := 15000,
	                               qx_Pulse => #tx_End15sPeriod);

	END_REGION

	REGION 3 - Add number of parcels in the register
	    //Each Region is used for different configurations

	    REGION 4.1 - When input counts are incrementing

	        IF #ix_IncrementingCounts THEN



	            //calculate new parcels per infeed
	            IF #s_infeed.diCounter >= #s_infeed.diLastScanCounter THEN
	                //Parcels are incremented normaly
	                #s_infeed.iNumberOfNewParcels := DINT_TO_INT(#s_infeed.diCounter - #s_infeed.diLastScanCounter);

	            ELSE
	                //Exception handling of parcel counter was reset in the partner PLC. Therefore for this scan we don't subtrack the ones of the previous scan
	                #s_infeed.iNumberOfNewParcels := DINT_TO_INT(#s_infeed.diCounter);
	            END_IF;

	            //Move current counter at the static variable of the last scan
	            #s_infeed.diLastScanCounter := #s_infeed.diCounter;

	            //add new parcels in the 1st register
	            #iq_InfeedArray.iCR[1] += (#s_infeed.iNumberOfNewParcels);
	        END_IF;

	    END_REGION

	    REGION 4.2 - When input counts are updated every 15 sec interval
	        //That logic here needs to be tested. There is a risk of loosing some parcels beacuse of the delay between the pLC to PLC communication.

	        IF NOT #ix_IncrementingCounts AND #tx_End15sPeriod THEN
	            #iq_InfeedArray.iCR[1] := DINT_TO_INT(#s_infeed.diCounter);
	        END_IF;
	    END_REGION

	END_REGION

	REGION 5 - Flow rate calculation
	    // The 15 second period has passed
	    IF (#tx_End15sPeriod) THEN


	        // Initialize static flow buffer
	        #s_infeed.diFlowRate30sec := L#0;
	        #s_infeed.diFlowRate1min := L#0;
	        #s_infeed.diFlowRate3min := L#0;
	        #s_infeed.diFlowRate10min := L#0;

	        // Loop through 40 Counting Registers per infeed
	        FOR #ti_LC_k := 1 TO 40 DO

	            // 30 sec flow handling
	            IF #ti_LC_k <= 2 THEN
	                #s_infeed.diFlowRate30sec += INT_TO_DINT(#iq_InfeedArray.iCR[#ti_LC_k]);

	                // Conversion to full hour
	                IF #ti_LC_k = 2
	                THEN
	                    #s_infeed.diFlowRate30sec *= L#120;
	                    //Normalise
	                    #s_infeed.diFlowRate30sec /= #sdi_AverageLength;

	                END_IF;
	            END_IF;

	            // 1 minute flow handling
	            IF #ti_LC_k <= 4 THEN
	                #s_infeed.diFlowRate1min += INT_TO_DINT(#iq_InfeedArray.iCR[#ti_LC_k]);

	                // Conversion to full hour
	                IF #ti_LC_k = 4 THEN
	                    #s_infeed.diFlowRate1min *= L#60;
	                    //Normalise
	                    #s_infeed.diFlowRate1min /= #sdi_AverageLength;
	                END_IF;
	            END_IF;

	            // 3 minutes flow handling
	            IF #ti_LC_k <= 12 THEN
	                #s_infeed.diFlowRate3min += INT_TO_DINT(#iq_InfeedArray.iCR[#ti_LC_k]);

	                // Conversion to full hour
	                IF #ti_LC_k = 12 THEN
	                    #s_infeed.diFlowRate3min *= L#20;
	                    //Normalise
	                    #s_infeed.diFlowRate3min /= #sdi_AverageLength;
	                END_IF;
	            END_IF;

	            // 10 minutes flow handling
	            #s_infeed.diFlowRate10min += INT_TO_DINT(#iq_InfeedArray.iCR[#ti_LC_k]);

	            // Conversion to full hour
	            IF #ti_LC_k = 40
	            THEN
	                #s_infeed.diFlowRate10min *= L#6;
	                //Normalise
	                #s_infeed.diFlowRate10min /= #sdi_AverageLength;
	            END_IF;

	        END_FOR;

	    END_IF;

	END_REGION

	REGION 6 - Cumulative flow at evaluation point

	    IF (#tx_End15sPeriod) THEN

	        //initialise static variable
	        #sdi_CumulativeFlowRate := L#0;

	        FOR #ti_LC_k := 1 TO 4 BY 1 DO

	            #sdi_CumulativeFlowRate += INT_TO_DINT(#iq_InfeedArray.iCR[#ti_LC_k]);

	        END_FOR;

	        // Conversion to full hour
	        #sdi_CumulativeFlowRate *= L#60;

	        //Normalise
	        #sdi_CumulativeFlowRate /= #sdi_AverageLength;

	    END_IF;

	END_REGION

	REGION 7 - Shift arrays when 15s flow period ends

	    // 15 seconds period elapsed
	    IF (#tx_End15sPeriod) THEN

	        // Shifted counting register by one element down
	        MOVE_BLK(IN := #iq_InfeedArray.iCR[1],
	                 COUNT := 59,
	                 OUT => #iq_InfeedArray.iCR[2]);

	        // Reset first registter
	        #iq_InfeedArray.iCR[1] := 0;


	    END_IF;

	END_REGION

	REGION 8 - Compare Current Value with Set Point

	    IF (#tx_End15sPeriod) THEN

	        IF #sdi_CumulativeFlowRate >= INT_TO_DINT(#iqUDT_FlowControlHMI.Setpoint) THEN

	            #si_CurrentConsecutivesAboveSP += 1;  //increment consecutives above set point
	            #si_CurrentConsecutivesBelowSP := 0;  //reset consecutives below set point
	        ELSE

	            #si_CurrentConsecutivesAboveSP := 0;  //reset consecutives above set point
	            #si_CurrentConsecutivesBelowSP += 1;  //increment consecutives below set point

	            //limit consecutives below set point to threshold value. Protection against INT overflow
	            IF #si_CurrentConsecutivesBelowSP >= 3 THEN

	                #si_CurrentConsecutivesBelowSP := 3;

	            END_IF;

	        END_IF;

	    END_IF;

	END_REGION

	REGION 9 - Evaluation - Apply flow control
	    //The evaluation period is specified by UPS at 1min or 4 intervals of 15 seconds

	    IF (#tx_End15sPeriod) AND #si_CurrentConsecutivesAboveSP > 0 THEN

	        //divide  current consecutives above SP with the number of intervals for evaluation ,,
	        #tr_quotient := INT_TO_REAL(#si_CurrentConsecutivesAboveSP) / INT_TO_REAL(4);

	        //call fraction to check the number of decimal places of the quotient
	        #tr_fraction := FRAC(#tr_quotient);

	        //If there are no decimal places then the current consecutive above set point is multiple
	        //of the evaluation period. Therefore the evaluation of the flow control should take place.
	        IF #tr_fraction = 0.0 THEN


	            REGION 9.1 - Request stop to limit flow

	                IF
	                    #s_infeed.Active                                      //infeed running / activated ..
	                    AND NOT #s_infeed.RequestStop                            // .. and not already stopped...
	                    AND NOT #s_infeed.DuringMinimumStopTime                  // .. and not during minimum time to stop

	                THEN
	                    #s_infeed.RequestStop := TRUE;
	                    #s_infeed.OneShotRequestStop := TRUE;
	                    //exit loop to stop one infeed every evaluation interval
	                END_IF;

	            END_REGION

	        END_IF;

	    END_IF;

	END_REGION

	REGION 10 - Evaluation - Remove flow control

	    IF (#tx_End15sPeriod) AND #si_CurrentConsecutivesBelowSP >= 3 THEN
	        #s_infeed.RequestStop := FALSE;
	    END_IF;

	END_REGION

	REGION 11  - Set minimum time of stopped time
	    //Set minimum time to stop 1min
	    #s_FB_MinStopTimeActive(iudi_OnDelayTime := 0,
	                            iudi_OffDelayTime := 60000,
	                            ix_SignalToDelay := #s_infeed.OneShotRequestStop,
	                            ix_Enable := TRUE,
	                            qx_DelayedSignal => #s_infeed.DuringMinimumStopTime);

	    //reset one shot request to stop
	    #s_infeed.OneShotRequestStop := FALSE;



	END_REGION

	REGION 12 - HMI Enable / Disable

	    //Command to disable frlow control from HMI
	    #sx_Disabled := #iqUDT_FlowControlHMI.CommandToDisable;

	END_REGION

	REGION 12 - Ouput the request stop

	    #qx_LimitFlowInfeed := (#s_infeed.RequestStop OR #s_infeed.DuringMinimumStopTime) AND NOT #sx_Disabled;

	END_REGION

	REGION 13 - Output flow rates

	    //Disabled status to HMI
	    #iqUDT_FlowControlHMI.DisabledStatus := #sx_Disabled;

	    ///Output 15 Sec interval one shot
	    #qx_New15SecInterval := #tx_End15sPeriod;

	    //Cumulative
	    #iqUDT_FlowControlHMI.CalculatedFlow := DINT_TO_INT(#sdi_CumulativeFlowRate);

	    //Infeed 1
	    #qdi_30secFlowInfeed := (#s_infeed.diFlowRate30sec);
	    #qdi_1minFlowInfeed := (#s_infeed.diFlowRate1min);
	    #qdi_3minFlowInfeed := (#s_infeed.diFlowRate3min);
	    #qdi_10minFlowInfeed := (#s_infeed.diFlowRate10min);

	END_REGION

END_FUNCTION_BLOCK

